// TwinCAT 3 PLC project control
// ProgramVersion: 3.1.4023.0
// libraries:
//   CmpBitmapPool, * (System)
//   Tc2_MC2, * (Beckhoff Automation GmbH)
//   Tc2_ModbusRTU, * (Beckhoff Automation GmbH)
//   Tc2_SerialCom, * (Beckhoff Automation GmbH)
//   Tc2_Standard, * (Beckhoff Automation GmbH)
//   Tc2_System, * (Beckhoff Automation GmbH)
//   Tc2_Utilities, * (Beckhoff Automation GmbH)
//   Tc3_Module, * (Beckhoff Automation GmbH)
//   VisuDialogs, * (System)
//   VisuSymbols,3.5.10.0,System
// project tree:
//   FB/ Rec_Ctrl.TcPOU
//   / GlobalTextList.TcGTLO, ImagePool_Base.TcIPO (not stored), PlcTask.TcTTO, Recipt_no.TcTLO, step.TcTLO, Visualization Manager.TcVMO (not stored), VISU_TASK.TcTTO
//   GVLs/ GVL.TcGVL
//   POUs/ MAIN.TcPOU, MOTION.TcPOU, POU.TcPOU
//   VISUs/ ALARM.TcVIS, IO_TABLE.TcVIS, MainBase.TcVIS, MOTION.TcVIS, PARAMETER.TcVIS, Recipt.TcVIS

CONFIGURATION control
    RESOURCE PLC ON TwinCAT3
        TASK PlcTask(INTERVAL := T#10ms, PRIORITY := 20);
        TASK VISU_TASK(INTERVAL := T#200000us, PRIORITY := 30);
        PROGRAM MAIN WITH PlcTask : MAIN;
        PROGRAM POU WITH PlcTask : POU;
        PROGRAM MOTION WITH PlcTask : MOTION;
        PROGRAM VisuElems_Visu_Prg WITH VISU_TASK : VisuElems.Visu_Prg;
    END_RESOURCE
END_CONFIGURATION

// ---- GVLs/GVL.TcGVL

VAR_GLOBAL
	

DI0_0 AT %I* :BOOL;
DI0_1 AT %I* :BOOL;
DI0_2 AT %I* :BOOL;
DI0_3 AT %I* :BOOL;
DI0_4 AT %I* :BOOL;
DI0_5 AT %I* :BOOL;
DI0_6 AT %I* :BOOL;
DI0_7 AT %I* :BOOL;

DI1_0 AT %I* :BOOL;
DI1_1 AT %I* :BOOL;
DI1_2 AT %I* :BOOL;
DI1_3 AT %I* :BOOL;
DI1_4 AT %I* :BOOL;
DI1_5 AT %I* :BOOL;
DI1_6 AT %I* :BOOL;
DI1_7 AT %I* :BOOL;

DI2_0 AT %I* :BOOL;
DI2_1 AT %I* :BOOL;
DI2_2 AT %I* :BOOL;
DI2_3 AT %I* :BOOL;
DI2_4 AT %I* :BOOL;
DI2_5 AT %I* :BOOL;
DI2_6 AT %I* :BOOL;
DI2_7 AT %I* :BOOL;

DI3_0 AT %I* :BOOL;
DI3_1 AT %I* :BOOL;
DI3_2 AT %I* :BOOL;
DI3_3 AT %I* :BOOL;
DI3_4 AT %I* :BOOL;
DI3_5 AT %I* :BOOL;
DI3_6 AT %I* :BOOL;
DI3_7 AT %I* :BOOL;


DO0_0 AT %Q* :BOOL;
DO0_1 AT %Q* :BOOL;
DO0_2 AT %Q* :BOOL;
DO0_3 AT %Q* :BOOL;
DO0_4 AT %Q* :BOOL;
DO0_5 AT %Q* :BOOL;
DO0_6 AT %Q* :BOOL;
DO0_7 AT %Q* :BOOL;

DO1_0 AT %Q* :BOOL;
DO1_1 AT %Q* :BOOL;
DO1_2 AT %Q* :BOOL;
DO1_3 AT %Q* :BOOL;
DO1_4 AT %Q* :BOOL:=1;
DO1_5 AT %Q* :BOOL:=1;
DO1_6 AT %Q* :BOOL:=1;
DO1_7 AT %Q* :BOOL:=1;

DO2_0 AT %Q* :BOOL;
DO2_1 AT %Q* :BOOL;
DO2_2 AT %Q* :BOOL;
DO2_3 AT %Q* :BOOL;
DO2_4 AT %Q* :BOOL;
DO2_5 AT %Q* :BOOL;
DO2_6 AT %Q* :BOOL;
DO2_7 AT %Q* :BOOL;

DO3_0 AT %Q* :BOOL;
DO3_1 AT %Q* :BOOL;
DO3_2 AT %Q* :BOOL;
DO3_3 AT %Q* :BOOL;
DO3_4 AT %Q* :BOOL;
DO3_5 AT %Q* :BOOL;
DO3_6 AT %Q* :BOOL;
DO3_7 AT %Q* :BOOL;

DO4_0 AT %Q* :BOOL;
DO4_1 AT %Q* :BOOL;
DO4_2 AT %Q* :BOOL;
DO4_3 AT %Q* :BOOL;
DO4_4 AT %Q* :BOOL;
DO4_5 AT %Q* :BOOL;
DO4_6 AT %Q* :BOOL;
DO4_7 AT %Q* :BOOL;

DO5_0 AT %Q* :BOOL;
DO5_1 AT %Q* :BOOL;
DO5_2 AT %Q* :BOOL;
DO5_3 AT %Q* :BOOL;
DO5_4 AT %Q* :BOOL;
DO5_5 AT %Q* :BOOL;
DO5_6 AT %Q* :BOOL;
DO5_7 AT %Q* :BOOL;


AI0_0 AT %I* :UINT;
AI0_1 AT %I* :UINT;
AI0_2 AT %I* :UINT;
AI0_3 AT %I* :UINT;//CG1

AI1_0 AT %I* :UINT;//CG2
AI1_1 AT %I* :UINT;//CG3
AI1_2 AT %I* :UINT;
AI1_3 AT %I* :UINT;

AI2_0 AT %I* :UINT;//temp new add
AI2_1 AT %I* :UINT;
AI2_2 AT %I* :UINT;
AI2_3 AT %I* :UINT;


AO0_0 AT %Q* :UINT;
AO0_1 AT %Q* :UINT;
AO0_2 AT %Q* :UINT;
AO0_3 AT %Q* :UINT;

GV1_CLS_DEVINP: BOOL;
GV1_OPN_DEVINP: BOOL;
GV1_OPN_CONST:REAL:=-10;

GV2_CLS_DEVINP: BOOL;
GV2_OPN_DEVINP: BOOL;
GV2_OPN_CONST:REAL:=10;

MFC1_open_btn:BOOL;
MFC2_open_btn:BOOL;

HTC_SetPos:WORD;
HTC_SetPr:WORD;
Rec_start_btn:BOOL;
Rec_stop_btn:BOOL;

//Recipt variable
lv80_btn: BOOL;
WSU_btn: BOOL;
MFC1_Inp: REAL;
MFC2_Inp: REAL;
GV1_btn_open: BOOL;
GV1_btn_close: BOOL;
GV2_btn_open: BOOL;
GV2_btn_close: BOOL;

SV1 : WORD;
SV2 : WORD;
SV3 : WORD;

Temp_Recipt_step: Recipt_step;

M1TOM2:BOOL;
M2ToM3:BOOL;
M3ToM2:BOOL;
M2ToM1:BOOL;
ON_POS:BOOL;
CUR_step_name:STRING(20);
Rec_finish:BOOL;
ON_POS_FLAG: BOOL;
M2ToM1_flag: BOOL;
M3ToM2_flag: BOOL;
M2ToM3_flag: BOOL;
M1ToM2_flag: BOOL;
swing_btn:BOOL;
take_up_btn:BOOL;
put_down_btn:BOOL;
Rec_take_up_finish:BOOL;
Rec_put_down_finish:BOOL;
M2_pressure_setting:REAL;
M2_current_pressure:real;
END_VAR

// ---- POUs/MAIN.TcPOU
PROGRAM MAIN
VAR
	MbMster: ModbusRtuMaster_KL6x22B;
	Mb_ID: BYTE;
	MbR_Q: WORD;
	MbR_Addr: WORD;
	Data_Read : ARRAY[1..8] OF INT;
	Data_Write : WORD;
	En_Read : BOOL;
    En_Write : BOOL;	
	MbW_Addr: WORD;
	
	PV1 : INT;
	PV2 : INT;
	PV3 : INT;
	
	
	
	nVar: INT;
	bVar1: BOOL;
	bVar3: BOOL;
	bVar2: BOOL;
	
	TTR91_U_CG1: LREAL;
	TTR91_P_CG1: LREAL;
	TTR91_C: REAL:=6.304;
	temp_CG1: LREAL;
	temp_string_CG1:STRING(255);
	strlen_CG1:INT;
	str1_CG1:STRING(255);
	str2_CG1:STRING(255);
	show_CG1:STRING(255);
	aSplit_CG1       : ARRAY[1..5] OF STRING(255);
	bResultSplit_CG1 : BOOL;
	i_CG1            : UDINT;
	
	TTR91_U_CG2: LREAL;
	TTR91_P_CG2: LREAL;
	temp_CG2: LREAL;
	temp_string_CG2:STRING(255);
	strlen_CG2:INT;
	str1_CG2:STRING(255);
	str2_CG2:STRING(255);
	show_CG2:STRING(255);
	aSplit_CG2       : ARRAY[1..5] OF STRING(255);
	bResultSplit_CG2 : BOOL;
	i_CG2            : UDINT;
	
	TTR91_U_CG3: LREAL;
	TTR91_P_CG3: LREAL;
	temp_CG3: LREAL;
	temp_string_CG3:STRING(255);
	strlen_CG3:INT;
	str1_CG3:STRING(255);
	str2_CG3:STRING(255);
	show_CG3:STRING(255);
	aSplit_CG3       : ARRAY[1..5] OF STRING(255);
	bResultSplit_CG3 : BOOL;
	i_CG3            : UDINT;
		

	ATM1_dis: REAL;
	ATM2_dis: REAL;
	ATM3_dis: REAL;
	MFC1_dis: REAL;
	MFC2_dis: REAL;
	
	MFC1_Out: UINT;
	MFC2_Out: uINT;
	
	

	
	WSU_DEVINP: BOOL;
	RST_BTN: BOOL;
	ALM_PUMP_COOL: BOOL;
	ALM_MFC1_DEV: BOOL;
	ALM_MFC2_DEV: BOOL;
	ALM_WATER_TEMP: BOOL;
	ALM_WATER_Prs: BOOL;
	ALM_Heater1_Temp:BOOL;
	ALM_Heater2_Temp:BOOL;
	ALM_Heater_cool:BOOL;
	ALM_GV1_Snr:BOOL;
	ALM_GV2_Snr:BOOL;
	ALM_inlet_prs:BOOL;
	
	MFC_ALM_TIMER1:TON;
	MFC_ALM_TIMER2:TON;
	WTR_TEMP_ALM_TIMER:TON;
	WP_IN_ALM_TIMER:Ton;
	WTR_DELTA_ALM_TIMER:Ton;
	HEATER_TEMP_ALM_TIMER1:Ton;
	HEATER_TEMP_ALM_TIMER2:Ton;
	
	MFC_ALM_TRIG1:R_TRIG;
	MFC_ALM_TRIG2:R_TRIG;
	WTR_TEMP_ALM_TRIG:R_TRIG;
	WP_IN_ALM_TRIG:R_TRIG;
	WTR_DELTA_ALM_TRIG:R_TRIG;
	HEATER_TEMP_ALM_TRIG1:R_TRIG;
	HEATER_TEMP_ALM_TRIG2:R_TRIG;
	
	MFC_ALM_FLAG1:BOOL;
	MFC_ALM_FLAG2:BOOL;
	WTR_TEMP_ALM_FLAG:BOOL;
	WP_IN_ALM_FLAG:BOOL;
	WTR_DELTA_ALM_FLAG:BOOL;
	HEATER_TEMP_ALM_FLAG1:BOOL;
	HEATER_TEMP_ALM_FLAG2:BOOL;
	
	
	MFC_delay:TIME;
	water_temp_delay:TIME;
	WP_IN_delay:TIME;
	WP_delta_delay:TIME;
	Heater_temp_delay:TIME;
	
	GV1_DFLAG: BOOL;
	GV1_TON: TON;
	ALM_GV1_CLS_SNR: BOOL;
	GV2_DFLAG: BOOL;
	GV2_TON: TON;
	ALM_GV2_CLS_SNR: BOOL;
	MbMster2: ModbusRtuMaster_KL6x22B;
	Data_Read2:ARRAY[1..8] OF INT;
	MbR_Q2: WORD;
	MbR_Addr2: WORD;
	En_Read2: BOOL;
	nVar2: INT;
	ADDR2: WORD; 
	En_Write2: BOOL;
	MbW_Addr2: WORD;
	Data_Write2: WORD;
	
	m3_up_btn:BOOL;
	m3_down_btn:BOOL;
	m3_rail_open:BOOL;
	m3_rail_cls:BOOL;
	m3_pin_up:BOOL;
	m3_pin_down:BOOL;
	
	m3_up_flag: BOOL;
	m3_down_flag: BOOL;
	up_step1: BOOL;
	up_step2: BOOL;
	M3_rail_opened: BOOL;
	up_step3: BOOL;
	up_step4: BOOL;
	up_step5: BOOL;
	down_step1: BOOL;
	down_step2: BOOL;
	down_step3: BOOL;
	down_step4: BOOL;
	M3_rail_closed: BOOL;
	HTC_ReadPos: INT;
	HTC_ReadPr: INT;
	//HTC_SetPr: WORD;
	HTC_MODE_Pr : BOOL;
	//HTC_SetPos: WORD;
	
	cur_mode:STRING(255);
	
	M1_sNR: BOOL;
	M2_SNR1: BOOL;
	M2_SNR2: BOOL;
	M3_SNR1: BOOL;
	M3_SNR2: BOOL;
	M3_SNR3: BOOL;
	mfc1_set: REAL;
	mfc2_set: REAL;
	M3_rail_CLOSE: BOOL;
	ATM1_STS: BOOL;
	ATM2_STS: BOOL;
	ATM3_STS: BOOL;
	LV80_STS: BOOL;
	WSU_STS: bool;
	TV_STS: BOOL;
	
	GetTime:NT_GetTime;
	cur_time:STRING(255);
	
	reset_btn:BOOL;
	insert_btn:bool;

	Rec_Ctrl:Rec_Ctrl;
	Copy_step:BOOL;
	Copy_recipe:BOOL;
	cur_step:INT:=1;
	cur_Rec:INT:=1;
	
	save_step_btn: BOOL;
	clear_step_btn:BOOL;
	//edit_step_btn:BOOL;	
	pre_step:INT:=1;
	pre_recipe:INT:=1;
	Rec_finish_delay: TON;
	Rec_finish_trig: R_TRIG;
	take_up_action: BOOL;
	put_down_action: BOOL;
	Rec_stop: BOOL;
	Rec_stop_btn_delay: TON;
	put_down_reset_action: TON;
	put_down_action_reset_in: BOOL;
	take_up_action_reset_in: BOOL;
	take_up_reset_action: TON;
	i: INT;
	j: INT;
	recipe_varible_reset_btn: BOOL;

	q: INT:=30;
	insert_delay:TON;
	insert_in:BOOL;
	insert_during: BOOL;
	insert_finish: BOOL;
END_VAR


VAR RETAIN
    MFC_delay_show:UINT;
	water_temp_delay_show:UINT;
	WP_IN_delay_show:UINT;
	WP_delta_delay_show:UINT;
	Heater_temp_delay_show:UINT;
	MFC_alarm_setting:REAL;
	water_temp_setting:REAL;
	WP_IN_setting:REAL;
	WP_delta_setting:REAL;
	Heater_temp_seeting:REAL;
	Full_recipt: ARRAY [1..10] OF One_Recipt;
END_VAR

CASE nVar OF 
     0 : 
		 En_Read := FALSE;
         En_Write := FALSE;	 
         IF NOT MbMster.BUSY AND NOT En_Write THEN
		   nVar := 1;	
		 END_IF
	 1 :
	     Mb_ID := 1;
		 MbR_Q := 1;
		 MbR_Addr := 130;
		 En_Read := TRUE;
         IF NOT MbMster.BUSY AND En_Read THEN
		   PV3 := MAIN.Data_Read[1]; 
		   nVar := 2;	
		 END_IF

     2 : 
	 
		 En_Read := FALSE;
         En_Write := FALSE;
         IF NOT MbMster.BUSY AND NOT En_Read  THEN
		   nVar := 3;	
		 END_IF
	 3 :
	     Mb_ID := 2;
		 MbR_Q := 1;
		 MbR_Addr := 130;
		 En_Read := TRUE;
         IF NOT MbMster.BUSY AND En_Read  THEN
		   PV1 := MAIN.Data_Read[1];				 
		   nVar := 4;	
		 END_IF	    
     4 : 

		 En_Read := FALSE;
         En_Write := FALSE;
         IF NOT MbMster.BUSY AND NOT En_Read  THEN
		   nVar := 5;	
		 END_IF
	 5 :
	     Mb_ID := 3;
		 MbR_Q := 1;
		 MbR_Addr := 130;
		 En_Read := TRUE;
         IF NOT MbMster.BUSY AND En_Read  THEN
		   PV2 := MAIN.Data_Read[1];			 
		   nVar := 6;	
		 END_IF	 
     6 : 
	 
         MAIN.Data_Write := SV1;		 
		 En_Read := FALSE;
         En_Write := FALSE;
         IF NOT MbMster.BUSY AND NOT En_Read  THEN
		   nVar := 7;	
		 END_IF
	 7 :
	     Mb_ID := 1;
		 MbW_Addr := 49;
		 En_Write := TRUE;
         IF NOT MbMster.BUSY AND En_Write  THEN
		   nVar := 8;	
		 END_IF
     8 : 
		 En_Read := FALSE;
         En_Write := FALSE;
         MAIN.Data_Write := SV2;		 
         IF NOT MbMster.BUSY  AND NOT En_Write  THEN
		   nVar := 9;	
		 END_IF
	 9 :
	     Mb_ID := 2;
		 MbW_Addr := 49;
		 En_Write := TRUE;
         IF NOT MbMster.BUSY  AND En_Write  THEN
		   nVar := 10;	
		 END_IF
     10 : 
		 En_Read := FALSE;
         En_Write := FALSE;
		 MAIN.Data_Write := SV3;
         IF NOT MbMster.BUSY  AND NOT En_Write  THEN
		   nVar := 11;	
		 END_IF
	 11 :
	     Mb_ID := 3;
		 MbW_Addr := 49;
		 En_Write := TRUE;
         IF NOT MbMster.BUSY  AND En_Write  THEN
		   nVar := 0;	
		 END_IF  	 


//ELSE 
		 //nVar := 0;
         //bVar1 := NOT bVar1; 
         //bVar2 := bVar1 OR bVar2; 
END_CASE;	


MbMster.ReadRegs(
	UnitID:= Mb_ID, 
	Quantity:= MbR_Q,
	MBAddr:= MbR_Addr, 
	cbLength:= SIZEOF(Data_Read), 
	pMemoryAddr:= ADR(Data_Read), 
	Execute:= En_Read, 
	Timeout:= T#10S, 
	BUSY=> , 
	Error=> , 
	ErrorId=> , 
	cbRead=> );

MbMster.WriteRegs(
	UnitID:= Mb_ID, 
	Quantity:= 1, 
	MBAddr:= MbW_Addr, 
	cbLength:= SIZEOF(Data_Write), 
	pMemoryAddr:= ADR(Data_Write), 
	Execute:= En_Write, 
	Timeout:= T#10S, 
	BUSY=> , 
	Error=> , 
	ErrorId=> , 
	cbRead=> );	
	
//============= RS485 CH2	

CASE nVar2 OF 
     0 : 
		 En_Read2 := FALSE;
         En_Write2 := FALSE;	 
         IF NOT MbMster2.BUSY  AND NOT En_Read2 THEN
		   nVar2 := 1;	
		 END_IF
	 1 :
	     //Mb_ID := 1;
		 MbR_Q2 := 1;
		 MbR_Addr2 := 263;//259;
		 En_Read2 := TRUE;
         IF NOT MbMster2.BUSY  AND   En_Read2 THEN
			 HTC_ReadPos := MAIN.Data_Read2[1];
		     nVar2 := 2;	
		 END_IF
	 2 : 
	   	 //MbW_Addr2 := WADDR2;
		 En_Read2 := FALSE;
		 En_Write2 := FALSE;
         IF NOT MbMster2.BUSY AND NOT En_Read2 THEN
		   nVar2 := 3;	
		 END_IF
	 3 :
	     //Mb_ID := 1;
		 //MbR_Q2 := 1;
		 IF HTC_MODE_Pr THEN
			HTC_SetPos :=0; 
		 END_IF
		 MAIN.Data_Write2 := HTC_SetPos;
		 MbW_Addr2 := 260;
		 En_Write2 := TRUE;
         IF NOT MbMster2.BUSY  AND   En_Write2 THEN
		     nVar2 := 4;	
		 END_IF
	 4 : 
	   	 //MbW_Addr2 := WADDR2;
		 En_Read2 := FALSE;
		 En_Write2 := FALSE;
         IF NOT MbMster2.BUSY AND NOT En_Write2 THEN
		   nVar2 := 5;	
		 END_IF		 		 
	 5 :
	     //Mb_ID := 1;
		 MbR_Q2 := 1;
		 MbR_Addr2 := 259;//263;
		 En_Read2 := TRUE;
         IF NOT MbMster2.BUSY  AND   En_Read2 THEN
			 HTC_ReadPr := MAIN.Data_Read2[1];
		     nVar2 := 6;	
		 END_IF
	 6 : 
	   	 //MbW_Addr2 := WADDR2;
		 En_Read2 := FALSE;
		 En_Write2 := FALSE;
         IF NOT MbMster2.BUSY AND NOT En_Read2 THEN
		   nVar2 := 7;	
		 END_IF
	 7 :
	     //Mb_ID := 1;
		 //MbR_Q2 := 1;
		 IF NOT HTC_MODE_Pr THEN
			 HTC_SetPr := 0;
		 END_IF
		 MAIN.Data_Write2 := HTC_SetPr;
		 MbW_Addr2 := 1123;
		 En_Write2 := TRUE;
         IF NOT MbMster2.BUSY  AND   En_Write2 THEN
		     nVar2 := 8;	
		 END_IF
	 8 : 
	   	 //MbW_Addr2 := WADDR2;
		 En_Read2 := FALSE;
		 En_Write2 := FALSE;
         IF NOT MbMster2.BUSY AND NOT En_Write2 THEN
		   nVar2 := 0;	
		 END_IF		 		 
		 
END_CASE;


MbMster2.ReadRegs(
	UnitID:= 1, 
	Quantity:= MbR_Q2, 
	MBAddr:= MbR_Addr2, 
	cbLength:= SIZEOF(Data_Read2), 
	pMemoryAddr:= ADR(Data_Read2), 
	Execute:= En_Read2, 
	Timeout:= T#10S, 
	BUSY=> , 
	Error=> , 
	ErrorId=> , 
	cbRead=> );

	MbMster2.WriteRegs(
	UnitID:= 1, 
	Quantity:= 1, 
	MBAddr:= MbW_Addr2, 
	cbLength:= SIZEOF(Data_Write2), 
	pMemoryAddr:= ADR(Data_Write2), 
	Execute:= En_Write2, 
	Timeout:= T#10S, 
	BUSY=> , 
	Error=> , 
	ErrorId=> , 
	cbRead=> );	


//=========================
CG1_trans();
CG2_trans();
CG3_trans();
interlock();
valve_control();
//ALARM();
snr_status();


IF insert_btn  = 1  THEN
	step_insert();
END_IF

IF insert_finish THEN
	insert_btn:=0;
	insert_finish:=0;
END_IF

IF Rec_stop_btn THEN
	Rec_stop:=1;
	REC_func();	
END_IF
Rec_stop_btn_delay(IN:=Rec_stop,PT:=T#0.1S,Q=>);
IF Rec_stop_btn_delay.Q THEN
	REC_func();	
	Rec_stop:=0;
	Rec_finish:=1;
END_IF

IF Rec_start_btn THEN
	REC_func();
END_IF

IF Rec_finish = 1 THEN
	Rec_reset();	
END_IF

IF Rec_finish_trig.Q THEN
	Rec_finish:=0;
END_IF

Rec_finish_delay(IN:=Rec_finish,PT:=T#0.1S,Q=>);
Rec_finish_trig(CLK:=Rec_finish_delay.Q,Q=>);

//ATM

	ATM1_dis:= 100*((UINT_TO_REAL(ai0_0)-19660)/13106);
	ATM2_dis:= 100*((UINT_TO_REAL(ai0_1)-19660)/13106);
	ATM3_dis:= 100*((UINT_TO_REAL(ai0_2)-19660)/13106);

//MFC1 1SLM  MFC 100SLM

    MFC1_dis:=1000*(UINT_TO_REAL(ai1_2)/32767);
	MFC2_dis:=100*(UINT_TO_REAL(ai1_3)/32767);	
	
	IF mfc1_open_btn THEN     //2022 0923 modify
		mfc1_set:=MFC1_Inp;
		ELSE
		mfc1_set:=0;
	END_IF
	
	IF mfc2_open_btn THEN
		mfc2_set:=MFC2_Inp;
		ELSE
		mfc2_set:=0;
	END_IF
	
	MFC1_Out:=REAL_TO_UINT(mfc1_set/1000*32767);
	MFC2_Out:=REAL_TO_UINT(mfc2_set/100*32767);
	ao0_2:=MFC1_Out;
    ao0_3:=MFC2_Out;
	
IF HTC_MODE_Pr = 1 THEN
	cur_mode:='Pos mode';
ELSE
	cur_mode:='Pr mode';
END_IF

IF GetTime.START AND NOT GetTime.BUSY THEN
	GetTime.START:=FALSE;
ELSE
	GetTime.START:=TRUE;
END_IF

GetTime(
	NETID:= '',
	START:= ,
	TMOUT:= ,
	BUSY=> ,
	ERR=>,
	ERRID=>,
	TIMESTR=>
);
cur_time:=CONCAT(WORD_TO_STRING(GetTime.TIMESTR.wHour),':');
cur_time:=CONCAT(cur_time,WORD_TO_STRING(GetTime.TIMESTR.wMinute));
cur_time:=CONCAT(cur_time,':');
cur_time:=CONCAT(cur_time,WORD_TO_STRING(GetTime.TIMESTR.wSecond));

IF save_step_btn THEN
	pre_step:=cur_step;
	pre_recipe:=cur_REC;
	Full_Recipt[cur_Rec].Rec_array[cur_step]:=Temp_Recipt_step;
END_IF

IF pre_step <> cur_step THEN
	Temp_Recipt_step:=Full_Recipt[cur_Rec].Rec_array[cur_step];
	pre_step:=cur_step;
END_IF

IF pre_recipe <> cur_REC THEN
	Temp_Recipt_step:=Full_Recipt[cur_Rec].Rec_array[cur_step];
	pre_recipe:=cur_rec;
END_IF

IF Copy_step AND cur_Step <> 1 THEN
	Temp_Recipt_step:=Full_Recipt[cur_Rec].Rec_array[cur_step-1];
END_IF

IF Copy_recipe AND cur_Rec <> 1 THEN
	Full_Recipt[cur_Rec]:=Full_Recipt[cur_Rec-1];
	Temp_Recipt_step:=Full_Recipt[cur_Rec].Rec_array[cur_step];
END_IF

IF clear_step_btn = 1 THEN
	Temp_Recipt_step.delay:=0;
	Temp_Recipt_step.GV1:=0;
	Temp_Recipt_step.GV2:=0;
	Temp_Recipt_step.LV80:=0;
	Temp_Recipt_step.M1toM2:=0;
	Temp_Recipt_step.M2_pressure_setting:=0;
	Temp_Recipt_step.M2toM1:=0;
	Temp_Recipt_step.M2toM3:=0;
	Temp_Recipt_step.M3_pressure_setting:=0;
	Temp_Recipt_step.M3toM2:=0;
	Temp_Recipt_step.MFC1_button:=0;
	Temp_Recipt_step.MFC1_Setting:=0;
	Temp_Recipt_step.MFC2_button:=0;
	Temp_Recipt_step.MFC2_Setting:=0;
	Temp_Recipt_step.NC1:=0;
	Temp_Recipt_step.NC2:=0;
	Temp_Recipt_step.NC3:=0;
	Temp_Recipt_step.NC4:=0;
	Temp_Recipt_step.NC5:=0;
	Temp_Recipt_step.NC6:=0;
	Temp_Recipt_step.NC7:=0;
	Temp_Recipt_step.NC8:=0;
	Temp_Recipt_step.NC9:=0;
	Temp_Recipt_step.Position_setting:=0;
	Temp_Recipt_step.RV1:=0;
	Temp_Recipt_step.RV2:=0;
	Temp_Recipt_step.Set2Pos:=0;
	Temp_Recipt_step.step_Name:='';
	Temp_Recipt_step.VENT2:=0;
	Temp_Recipt_step.WSU251:=0;
	Temp_Recipt_step.Swing:=0;
	Temp_Recipt_step.Take_up:=0;
	Temp_Recipt_step.Put_down:=0;
	Temp_Recipt_step.VB4:=0;
	Temp_Recipt_step.VENT3:=0;
END_IF
(*
IF edit_step_btn THEN
	Temp_Recipt_step:=Full_Recipt[cur_Rec].Rec_array[cur_step];
END_IF
*)

IF Rec_stop_btn THEN
	Rec_start_btn:=0;
END_IF

IF recipe_varible_reset_btn THEN
	Recipe_variable_reset();
END_IF

M2_current_pressure:=ATM1_dis;

ACTION ALARM:
//PUMP COOLING WATER

IF DO3_6 AND NOT di1_4 THEN	
	ALM_PUMP_COOL:=1;
END_IF



// inlet pressure

IF NOT di1_7 THEN 
	ALM_inlet_prs:=1;
	ELSE
	ALM_inlet_prs:=0;	
END_IF



//GV1
IF GV1_btn_close THEN
	GV1_DFLAG:=1;
END_IF

GV1_TON(IN:=GV1_DFLAG,PT:=T#3S,Q=>,ET=>);
IF GV1_TON.Q AND NOT DI2_0 THEN
	ALM_GV1_CLS_SNR:=1;
END_IF

IF GV1_btn_OPEN THEN
	GV1_DFLAG:=0;
END_IF


//GV2

IF GV2_btn_close THEN
	GV2_DFLAG:=1;
END_IF

GV2_TON(IN:=GV2_DFLAG,PT:=T#3S,Q=>,ET=>);
IF GV2_TON.Q AND NOT DI2_2 THEN
	ALM_GV2_CLS_SNR:=1;
END_IF

IF GV2_btn_OPEN THEN
	GV2_DFLAG:=0;
END_IF



//Light Tower

IF ALM_PUMP_COOL OR ALM_inlet_prs OR ALM_GV1_CLS_SNR OR ALM_GV2_CLS_SNR THEN
	DO1_4:=0;
	DO1_7:=0;
END_IF



// RST BUTTON
IF RST_BTN THEN
	DO1_4:=1;
	DO1_7:=1;
	ALM_PUMP_COOL:=0;
	ALM_inlet_prs:=0;
	ALM_GV1_CLS_SNR:=0;
	ALM_GV2_CLS_SNR:=0;
END_IF

//alarm delay setting
MFC_delay:=UINT_TO_TIME(MFC_delay_show)*1000;
water_temp_delay:=UINT_TO_TIME(water_temp_delay_show)*1000;
WP_IN_delay:=UINT_TO_TIME(WP_IN_delay_show)*1000;
WP_delta_delay:=UINT_TO_TIME(WP_delta_delay_show)*1000;
Heater_temp_delay:=UINT_TO_TIME(Heater_temp_delay_show)*1000;

MFC_ALM_TIMER1(IN:=MFC_ALM_FLAG1,PT:=MFC_delay,Q=>);
MFC_ALM_TIMER2(IN:=MFC_ALM_FLAG2,PT:=MFC_delay,Q=>);
WTR_TEMP_ALM_TIMER(IN:=WTR_TEMP_ALM_FLAG,PT:=water_temp_delay,Q=>);
WP_IN_ALM_TIMER(IN:=WP_IN_ALM_FLAG,PT:=WP_IN_delay,Q=>);
WTR_DELTA_ALM_TIMER(IN:=WTR_DELTA_ALM_FLAG,PT:=WP_delta_delay,Q=>);
HEATER_TEMP_ALM_TIMER1(IN:=HEATER_TEMP_ALM_FLAG1,PT:=Heater_temp_delay,Q=>);
HEATER_TEMP_ALM_TIMER2(IN:=HEATER_TEMP_ALM_FLAG2,PT:=Heater_temp_delay,Q=>);

MFC_ALM_TRIG1(CLK:=MFC_ALM_TIMER1.Q,Q=>);
MFC_ALM_TRIG2(CLK:=MFC_ALM_TIMER2.Q,Q=>);
WTR_TEMP_ALM_TRIG(CLK:=WTR_TEMP_ALM_TIMER.Q,Q=>);
WP_IN_ALM_TRIG(CLK:=WP_IN_ALM_TIMER.Q,Q=>);
WTR_DELTA_ALM_TRIG(CLK:=WTR_DELTA_ALM_TIMER.Q,Q=>);
HEATER_TEMP_ALM_TRIG1(CLK:=HEATER_TEMP_ALM_TIMER1.Q,Q=>);
HEATER_TEMP_ALM_TRIG2(CLK:=HEATER_TEMP_ALM_TIMER2.Q,Q=>);

IF (MFC1_Inp < MFC1_dis *(1-MFC_alarm_setting*0.01) OR MFC1_Inp > MFC1_dis *(1+MFC_alarm_setting*0.01)) AND MFC1_Inp <> 0 THEN
	MFC_ALM_FLAG1:=1;
	ALM_MFC1_DEV:=1;
ELSE
	MFC_ALM_FLAG1:=0;
	ALM_MFC1_DEV:=0;
END_IF

IF (MFC2_Inp < MFC2_dis *(1-MFC_alarm_setting*0.01) OR MFC2_Inp > MFC2_dis *(1+MFC_alarm_setting*0.01)) AND MFC2_Inp <> 0 THEN
	MFC_ALM_FLAG2:=1;
	ALM_MFC2_DEV:=1;
ELSE
	MFC_ALM_FLAG2:=0;
	ALM_MFC2_DEV:=0;
END_IF

IF MFC_ALM_TRIG1.Q OR MFC_ALM_TRIG2.Q THEN
	DO1_7:=0;//DO1_7:=0會叫
END_IF


IF PV1 > Heater_temp_seeting THEN
	HEATER_TEMP_ALM_FLAG1:=1;
	ALM_Heater1_Temp:=1;
ELSE
	HEATER_TEMP_ALM_FLAG1:=0;
	ALM_Heater1_Temp:=0;
END_IF

IF PV2 > Heater_temp_seeting THEN
	HEATER_TEMP_ALM_FLAG2:=1;
	ALM_Heater2_Temp:=1;
ELSE
	HEATER_TEMP_ALM_FLAG2:=0;
	ALM_Heater2_Temp:=0;
END_IF

IF HEATER_TEMP_ALM_TRIG1.Q OR HEATER_TEMP_ALM_TRIG2.Q THEN
	DO1_7:=0;
END_IF
END_ACTION

ACTION CG1_trans:
TTR91_U_CG1 := AI0_3/6553.5 ;
temp_CG1 := (TTR91_U_CG1 - TTR91_C)/1.286;
TTR91_P_CG1 := EXPT(10,temp_CG1);
IF TTR91_P_CG1 > 1 THEN
	temp_string_CG1 := LREAL_TO_STRING(TTR91_P_CG1);
	aSplit_CG1[1] := temp_string_CG1;
	FOR i_CG1:=1 TO 5 DO
    bResultSplit_CG1 := FindAndSplitChar( sSeparatorChar := '.',  pSrcString := ADR(aSplit_CG1[i_CG1]), 
                                      pLeftString    := ADR(aSplit_CG1[i_CG1]),   nLeftSize  := SIZEOF(aSplit_CG1[i_CG1]), 
                                      pRightString   := ADR(aSplit_CG1[i_CG1+1]), nRightSize := SIZEOF(aSplit_CG1[i_CG1+1]),
                                      bSearchFromRight := FALSE );
    IF NOT bResultSplit_CG1 THEN
        EXIT;
    END_IF
	END_FOR
	str2_CG1:=left(temp_string_CG1,3);
	IF TTR91_P_CG1 >= 100 THEN
		str2_CG1:=REAL_TO_STRING(STRING_TO_INT(str2_CG1)/100.0);
	ELSIF TTR91_P_CG1 < 100 AND TTR91_P_CG1 >= 10 THEN
		str2_CG1:=REAL_TO_STRING(STRING_TO_INT(str2_CG1)/10.0);
	ELSIF TTR91_P_CG1 >=1 AND TTR91_P_CG1 < 10 THEN
		str2_CG1:=REAL_TO_STRING(STRING_TO_real(str2_CG1));
	END_IF
	
	str1_CG1:=CONCAT('e+',INT_TO_STRING(len(aSplit_CG1[1])-1));
	show_CG1 := CONCAT (str2_CG1,str1_CG1);
ELSE
	temp_string_CG1 := LREAL_TO_STRING(TTR91_P_CG1);
	str1_CG1:=right(temp_string_CG1,3);
	str2_CG1:=left(temp_string_CG1,4);
	show_CG1 := CONCAT (str2_CG1,str1_CG1);
END_IF
END_ACTION

ACTION CG2_trans:
TTR91_U_CG2 := AI1_0/6553.5 ;
temp_CG2 := (TTR91_U_CG2 - TTR91_C)/1.286;
TTR91_P_CG2 := EXPT(10,temp_CG2);
IF TTR91_P_CG2 > 1 THEN
	temp_string_CG2 := LREAL_TO_STRING(TTR91_P_CG2);
	aSplit_CG2[1] := temp_string_CG2;
	FOR i_CG2:=1 TO 5 DO
    bResultSplit_CG2 := FindAndSplitChar( sSeparatorChar := '.',  pSrcString := ADR(aSplit_CG2[i_CG2]), 
                                      pLeftString    := ADR(aSplit_CG2[i_CG2]),   nLeftSize  := SIZEOF(aSplit_CG2[i_CG2]), 
                                      pRightString   := ADR(aSplit_CG2[i_CG2+1]), nRightSize := SIZEOF(aSplit_CG2[i_CG2+1]),
                                      bSearchFromRight := FALSE );
    IF NOT bResultSplit_CG2 THEN
        EXIT;
    END_IF
	END_FOR
	str2_CG2:=left(temp_string_CG2,3);
	IF TTR91_P_CG2 >= 100 THEN
		str2_CG2:=REAL_TO_STRING(STRING_TO_INT(str2_CG2)/100.0);
	ELSIF TTR91_P_CG2 < 100 AND TTR91_P_CG2 >=10 THEN
		str2_CG2:=REAL_TO_STRING(STRING_TO_INT(str2_CG2)/10.0);
	ELSIF TTR91_P_CG2 <10 AND TTR91_P_CG2 >=1 THEN
		 str2_CG2:=REAL_TO_STRING(STRING_TO_REAL(str2_CG2));
	END_IF
	
	str1_CG2:=CONCAT('e+',INT_TO_STRING(len(aSplit_CG2[1])-1));
	show_CG2 := CONCAT (str2_CG2,str1_CG2);
ELSE
	temp_string_CG2 := LREAL_TO_STRING(TTR91_P_CG2);
	str1_CG2:=right(temp_string_CG2,3);
	str2_CG2:=left(temp_string_CG2,4);
	show_CG2 := CONCAT (str2_CG2,str1_CG2);
END_IF
END_ACTION

ACTION CG3_trans:
TTR91_U_CG3 := AI1_1/6553.5 ;
temp_CG3 := (TTR91_U_CG3 - TTR91_C)/1.286;
TTR91_P_CG3 := EXPT(10,temp_CG3);
IF TTR91_P_CG3 > 1 THEN
	temp_string_CG3 := LREAL_TO_STRING(TTR91_P_CG3);
	aSplit_CG3[1] := temp_string_CG3;
	FOR i_CG3:=1 TO 5 DO
    bResultSplit_CG3 := FindAndSplitChar( sSeparatorChar := '.',  pSrcString := ADR(aSplit_CG3[i_CG3]), 
                                      pLeftString    := ADR(aSplit_CG3[i_CG3]),   nLeftSize  := SIZEOF(aSplit_CG3[i_CG3]), 
                                      pRightString   := ADR(aSplit_CG3[i_CG3+1]), nRightSize := SIZEOF(aSplit_CG3[i_CG3+1]),
                                      bSearchFromRight := FALSE );
    IF NOT bResultSplit_CG3 THEN
        EXIT;
    END_IF
	END_FOR
	str2_CG3:=left(temp_string_CG3,3);
	IF TTR91_P_CG3 >= 10 AND TTR91_P_CG3 < 100 THEN
		str2_CG3:=REAL_TO_STRING(STRING_TO_INT(str2_CG3)/10.0);
	ELSIF TTR91_P_CG3 >= 100 THEN
		str2_CG3:=REAL_TO_STRING(STRING_TO_INT(str2_CG3)/100.0);
	ELSIF TTR91_P_CG3 < 10 AND TTR91_P_CG3 >= 1 THEN
		str2_CG3:=REAL_TO_STRING(STRING_TO_REAL(str2_CG3));
	END_IF
	
	str1_CG3:=CONCAT('e+',INT_TO_STRING(len(aSplit_CG3[1])-1));
	show_CG3 := CONCAT (str2_CG3,str1_CG3);
ELSE
	temp_string_CG3 := LREAL_TO_STRING(TTR91_P_CG3);
	str1_CG3:=right(temp_string_CG3,3);
	str2_CG3:=left(temp_string_CG3,4);
	show_CG3 := CONCAT (str2_CG3,str1_CG3);
END_IF
END_ACTION

ACTION INTERLOCK:
//GV1

IF NOT DI0_0 AND NOT DI0_1 THEN
	GV1_CLS_DEVINP:=1;
	ELSE
	GV1_CLS_DEVINP:=0;	
END_IF

IF ATM1_DIS <GV1_OPN_CONST THEN
	GV1_OPN_DEVINP:=1;
	ELSE
	GV1_OPN_DEVINP:=0;	
END_IF

//GV2

IF NOT DI0_2 AND NOT DI0_3 THEN
	GV2_CLS_DEVINP:=1;
	ELSE
	GV2_CLS_DEVINP:=0;	
END_IF

IF ABS(ATM1_DIS-ATM2_DIS)>GV2_OPN_CONST THEN
	GV2_OPN_DEVINP:=1;
	ELSE
	GV2_OPN_DEVINP:=0;	
END_IF

// LV80 Pump

IF LV80_btn AND di1_4 THEN
	DO3_6:=1;
	ELSE
	DO3_6:=0;
	LV80_btn:=0;
END_IF

IF WSU_btn AND DO3_6 THEN
	DO3_7:=1;
	ELSE
	DO3_7:=0;	
END_IF

//wsu_devinp

IF DO3_6 THEN
	WSU_DEVINP:=0;
	ELSE
	WSU_DEVINP:=1;	
END_IF
END_ACTION

ACTION REC_func:
Rec_Ctrl(
	Enable		:= Rec_start_btn,
	Stop        := Rec_stop, 
	Step		:= Full_Recipt[cur_rec], 
	bStart		=> , 
	State       => , 
	bBusy		=> , 
	bDone		=> , 
	bError		=> );
END_ACTION

ACTION Rec_reset:
CUR_step_name:='';
GV1_btn_open:=0;
GV1_btn_close:=0;
GV2_btn_open:=0;
GV2_btn_close:=0;
lv80_btn:=0;
WSU_btn:=0;
MFC1_Inp:=0;
MFC2_Inp:=0;
mfc1_open_btn:=0;
mfc2_open_btn:=0;
DO2_0:=0;
DO2_1:=0;
DO2_2:=0;
DO2_3:=0;
DO2_4:=0;
DO2_5:=0;
DO2_6:=0;
DO2_7:=0;
DO3_0:=0;
DO3_1:=0;
DO3_2:=0;
DO3_3:=0;
DO4_0:=0;
DO4_1:=0;
DO4_2:=0;
DO4_3:=0;
DO4_4:=0;
DO4_5:=0;
DO4_6:=0;
DO4_7:=0;
DO5_0:=0;
ON_POS:=0;
M1TOM2:=0;
M2ToM3:=0;
M3ToM2:=0;
M2ToM1:=0;
ON_POS_FLAG:=0;
M1ToM2_flag:=0;
M2ToM3_flag:=0;
M3ToM2_flag:=0;
M2ToM1_flag:=0;
take_up_btn:=0;
put_down_btn:=0;
swing_btn:=0;
Rec_take_up_finish:=0;
Rec_put_down_finish:=0;
END_ACTION

ACTION Recipe_variable_reset:
FOR i := 1 TO 10 DO
	FOR j := 1 TO 30 DO
		Full_recipt[i].Rec_array[j].step_Name:= WSTRING_TO_STRING("");
		Full_recipt[i].Rec_array[j].GV1:=0;
		Full_recipt[i].Rec_array[j].GV2:=0;
		Full_recipt[i].Rec_array[j].LV80:=0;
		Full_recipt[i].Rec_array[j].M1toM2:=0;
		Full_recipt[i].Rec_array[j].M2_pressure_setting:=0;
		Full_recipt[i].Rec_array[j].M2toM1:=0;
		Full_recipt[i].Rec_array[j].M2toM3:=0;
		Full_recipt[i].Rec_array[j].M3toM2:=0;
		Full_recipt[i].Rec_array[j].MFC1_button:=0;
		Full_recipt[i].Rec_array[j].MFC1_Setting:=0;
		Full_recipt[i].Rec_array[j].MFC2_button:=0;
		Full_recipt[i].Rec_array[j].MFC2_Setting:=0;
		Full_recipt[i].Rec_array[j].NC1:=0;
		Full_recipt[i].Rec_array[j].NC2:=0;
		Full_recipt[i].Rec_array[j].NC3:=0;
		Full_recipt[i].Rec_array[j].NC4:=0;
		Full_recipt[i].Rec_array[j].NC5:=0;
		Full_recipt[i].Rec_array[j].NC6:=0;
		Full_recipt[i].Rec_array[j].NC7:=0;
		Full_recipt[i].Rec_array[j].NC8:=0;
		Full_recipt[i].Rec_array[j].NC9:=0;
		Full_recipt[i].Rec_array[j].Position_setting:=0;
		Full_recipt[i].Rec_array[j].Put_down:=0;
		Full_recipt[i].Rec_array[j].RV1:=0;
		Full_recipt[i].Rec_array[j].RV2:=0;
		Full_recipt[i].Rec_array[j].Set2Pos:=0;
		Full_recipt[i].Rec_array[j].Swing:=0;
		Full_recipt[i].Rec_array[j].Take_up:=0;
		Full_recipt[i].Rec_array[j].VB4:=0;
		Full_recipt[i].Rec_array[j].VENT3:=0;
		Full_recipt[i].Rec_array[j].VENT2:=0;
		Full_recipt[i].Rec_array[j].WSU251:=0;
	END_FOR
	
END_FOR
END_ACTION

ACTION SNR_STATUS:
M1_SNR:=NOT DI0_0;
M2_SNR1:=NOT DI0_1;
M2_SNR2:=NOT DI0_2;
M3_SNR1:=NOT DI0_3;
M3_SNR2:=NOT DI0_4;
M3_SNR3:=NOT DI0_5;

IF ATM1_dis > -10 THEN
	ATM1_STS:=1;
ELSE
	ATM1_STS:=0;
END_IF

IF ATM2_dis > -10 THEN
	ATM2_STS:=1;
ELSE
	ATM2_STS:=0;
END_IF

IF ATM3_dis > -10 THEN
	ATM3_STS:=1;
ELSE
	ATM3_STS:=0;
END_IF

IF DO3_6 THEN
	LV80_STS:=1;
ELSE
	LV80_STS:=0;
END_IF

IF DO3_7 THEN
	WSU_STS:=1;
ELSE
	WSU_STS:=0;
END_IF

IF HTC_ReadPos > 0 THEN
	TV_STS:=1;
ELSE
	TV_STS:=0;
END_IF
END_ACTION

ACTION step_insert:
insert_delay(IN:=insert_in,PT:=T#1MS,Q=>);

IF insert_in = 0 THEN
	insert_in:=1;
END_IF

IF insert_delay.Q AND q > cur_step THEN
	Full_Recipt[cur_Rec].Rec_array[q]:=Full_Recipt[cur_Rec].Rec_array[q-1];
	q:=q-1;
	insert_in:=0;	
END_IF

IF q = cur_step THEN
	Full_Recipt[cur_Rec].Rec_array[cur_step]:=Temp_Recipt_step;
	q:=30;
	insert_finish:=1;
END_IF
END_ACTION

ACTION valve_control:
//GV1 GV2

  IF GV1_btn_open THEN
	  DO1_0:=0;
	  DO1_1:=1;
  END_IF
  
 IF GV1_btn_close THEN
	  DO1_0:=1;
	  DO1_1:=0;
  END_IF 
  
   IF GV2_btn_open THEN
	  DO1_2:=0;
	  DO1_3:=1;
  END_IF
  
 IF GV2_btn_close THEN
	  DO1_2:=1;
	  DO1_3:=0;
  END_IF 
  
  // M3 LOAD 2022/09/23
  
	IF M3_rail_open THEN
	  DO0_0:=0;
	  DO0_1:=1;
	  DO0_4:=0;
	  DO0_5:=1;
	END_IF	 
	
	IF M3_rail_CLOSE THEN  
	  DO0_0:=1;
	  DO0_1:=0;
	  DO0_4:=1;
	  DO0_5:=0;
	END_IF	  
	
	IF M3_pin_up THEN
	  DO0_6:=1;
	  DO0_7:=0;
	  END_IF
	IF M3_pin_DOWN THEN  
	  DO0_6:=0;
	  DO0_7:=1;	  
	END_IF	  

	
	IF di2_5 AND di2_7 AND di3_1 AND di3_3 THEN
		M3_rail_opened:=1;
		ELSE
		M3_rail_opened:=0;	
	END_IF
		IF di2_4 AND di2_6 AND di3_0 AND di3_2 THEN
		M3_rail_closed:=1;
		ELSE
		M3_rail_closed:=0;	
	END_IF 

// up sequence 

 IF m3_up_btn OR (take_up_btn AND NOT take_up_action) THEN
    m3_up_flag:=1;
    m3_down_flag:=0;
    up_step1:=1;
	take_up_action:=1;
 END_IF
 IF m3_up_flag AND up_step1 THEN
    M3_rail_open:=1;
    up_step1:=0;
    up_step2:=1;
 END_IF
 IF m3_up_flag AND up_step2 AND M3_rail_opened THEN
    M3_pin_up:=1;
    up_step2:=0;
    up_step3:=1;
 END_IF
 IF m3_up_flag AND up_step3 AND di3_4 THEN
      M3_rail_open:=0;
   M3_rail_close:=1;//close M3 rail
   up_step3:=0;
   up_step4:=1;
 END_IF
 
 IF m3_up_flag AND up_step4 AND M3_rail_closed  THEN
      M3_pin_up:=0;
   M3_pin_DOWN:=1; // ADD BY HUGO
   up_step4:=0;
   up_step5:=1;
 END_IF
 IF  m3_up_flag AND up_step5 AND  di3_5 THEN
  M3_rail_close:=0;
  up_step5:=0;
  M3_pin_DOWN:=0;
  m3_up_flag:=0;  // ADD BY HUGO
  IF take_up_btn THEN
	  Rec_take_up_finish:=1;
  END_IF
  take_up_action_reset_in:=1;
 END_IF
take_up_reset_action(IN:=take_up_action_reset_in,PT:=T#0.15S,Q=>);
IF take_up_reset_action.Q THEN
	take_up_action:=0;
	take_up_action_reset_in:=0;
END_IF

 
//down sequence
 
 IF (m3_down_btn OR put_down_btn) AND NOT put_down_action THEN
    m3_up_flag:=0;
    m3_down_flag:=1;
    down_step1:=1;
	put_down_action:=1;
 END_IF
 
 IF m3_down_flag AND down_step1 THEN
    M3_pin_up:=1;
    down_step1:=0;
    down_step2:=1;
 END_IF
 
 IF m3_down_flag AND down_step2 AND di3_4 THEN
    M3_rail_open:=1;
    down_step2:=0;
    down_step3:=1;
 END_IF
 IF m3_down_flag AND down_step3 AND m3_rail_opened THEN
    M3_pin_up:=0;
     M3_pin_DOWN:=1; // ADD BY HUGO
    down_step3:=0;
    down_step4:=1;
 END_IF
 IF m3_down_flag AND down_step4 AND di3_5 THEN
    M3_rail_open:=0;
    down_step4:=0;
    m3_down_flag:=0; // ADD BY HUGO
    M3_pin_DOWN:=0;
	IF put_down_btn THEN
		Rec_put_down_finish:=1;
	END_IF
	put_down_action_reset_in:=1;
 END_IF
	
put_down_reset_action(IN:=put_down_action_reset_in,PT:=T#0.15S,Q=>);

IF put_down_reset_action.Q = 1 THEN
	put_down_action:=0;
	put_down_action_reset_in:=0;
END_IF
//reset

IF reset_btn = 1 THEN
	m3_up_btn:=0;
	m3_down_btn:=0;
	m3_down_flag:=0;
	m3_up_flag:=0;
	up_step1:=0;
	up_step2:=0;
	up_step3:=0;
	up_step4:=0;
	up_step5:=0;
	down_step1:=0;
	down_step2:=0;
	down_step3:=0;
	down_step4:=0;
	put_down_action:=0;
	take_up_action:=0;
END_IF

(*	
// up sequence	

	IF m3_up_btn THEN
	   m3_up_flag:=1;
	   m3_down_flag:=0;
	   up_step1:=1;
	END_IF
	IF m3_up_flag AND up_step1 THEN
	   M3_rail_open:=1;
	   up_step1:=0;
	   up_step2:=1;
	END_IF
	IF m3_up_flag AND up_step2 AND M3_rail_opened THEN
	   M3_pin_up:=1;
	   up_step2:=0;
	   up_step3:=1;
	END_IF
	IF m3_up_flag AND up_step3 AND di3_4 THEN
	     M3_rail_open:=0;
		 M3_rail_close:=1;//close M3 rail
		 up_step3:=0;
		 up_step4:=1;
	END_IF
	
	IF m3_up_flag AND up_step4 AND M3_rail_closed  THEN
	     M3_pin_up:=0;
		 up_step4:=0;
		 up_step5:=1;
	END_IF
	IF  m3_up_flag AND up_step5 AND  di3_5 THEN
		M3_rail_close:=0;
		M3_rail_closed:=0;
		up_step5:=0;
	END_IF
	
//down sequence
	
	IF m3_down_btn THEN
	   m3_up_flag:=0;
	   m3_down_flag:=1;
	   down_step1:=1;
	END_IF
	
	IF m3_down_flag AND down_step1 THEN
	   M3_pin_up:=1;
	   down_step1:=0;
	   down_step2:=1;
	END_IF
	
	IF m3_down_flag AND down_step2 AND di3_4 THEN
	   M3_rail_open:=1;
	   down_step2:=0;
	   down_step3:=1;
	END_IF
	IF m3_down_flag AND down_step3 AND m3_rail_opened THEN
	   M3_pin_up:=0;
	   down_step3:=0;
	   down_step4:=1;
	END_IF
	IF m3_down_flag AND down_step4 AND di3_5 THEN
	  down_step4:=0;
    END_IF 
*)
END_ACTION

END_PROGRAM

// ---- FB/Rec_Ctrl.TcPOU
FUNCTION_BLOCK Rec_Ctrl
VAR_INPUT
	Enable     : BOOL;
	Stop       : BOOL;
	Step	   :One_Recipt;
END_VAR
VAR_OUTPUT
	bStart : BOOL;
	bBusy  : BOOL;
	bDone  : BOOL;
	bError : BOOL;
	State  : INT;
END_VAR
VAR
	bTon : BOOL;
	dur : Ton;
	Rec_duration:Ton;
	nState: INT;
	i : INT := 1;
	pos_delay:TON;
	
	M2toM1_delay: Ton;
	M2toM1_in: BOOL;
END_VAR

IF Stop THEN
	bStart := FALSE;
	bBusy  := FALSE;
	bDone  := FALSE;
	bError := FALSE;
	bTon   := FALSE;
	nState := 0;
	i      := 1;
	Rec_finish:=1;
	Stop:=0;
END_IF



CASE nState OF
0 :	
	IF Enable AND NOT (bBusy OR bError) THEN
		bDone  := FALSE;
		bBusy  := TRUE;
		nState := 1;
		i      := 1;
	END_IF
	
	IF NOT Enable THEN
		bBusy  := FALSE;
		bError := FALSE;		
	END_IF	
1 :
	
	IF step.Rec_array[i].delay > 0 THEN //use delay to change step
		bTon   := TRUE;
		bStart := TRUE;	
		
	ELSIF step.Rec_array[i].Set2Pos = 1 THEN //wait until go to right place
		IF (step.Rec_array[i].M1toM2 OR step.Rec_array[i].M3toM2) AND MAIN.M2_SNR1 AND MAIN.M2_SNR2 THEN
			GVL.ON_POS:=1;
		END_IF
		
		IF step.Rec_array[i].M2toM3 AND MAIN.M3_SNR1 AND MAIN.M3_SNR2 THEN
			GVL.ON_POS:=1;
		END_IF
		
		IF step.Rec_array[i].M2toM1 AND main.M2_SNR1 = 0 AND main.M2_SNR2 = 0 THEN
			M2ToM1_in := 1;
			IF M2ToM1_delay.Q THEN
				ON_POS:=1;
			END_IF
		END_IF
		
		IF (Rec_take_up_finish AND take_up_btn) OR (Rec_put_down_finish AND put_down_btn) THEN
			ON_POS:=1;
		END_IF
		
		IF pos_delay.Q THEN
			Rec_take_up_finish:=0;
			Rec_put_down_finish:=0;
			ON_POS:=0;
			M2ToM1_in:=0;
			i:= i + 1;
			nState := 2;
		END_IF
		
	ELSIF step.Rec_array[i].M2_pressure_setting <> 0 THEN
		IF M2_current_pressure > step.Rec_array[i].M2_pressure_setting THEN
			i:= i + 1;
			nState := 2;
		END_IF
		
	ELSE
		i := i + 1;
		IF i > 30 THEN
			i := 1;
			Rec_start_btn:=0;
			Rec_finish:=1;
		END_IF		
	END_IF
	
	IF Rec_duration.Q  AND step.Rec_array[i].Set2Pos = 0 THEN
		i := i + 1;
		IF i > 30 THEN
			i := 1;
		END_IF
		nState := 2;
	END_IF

2 :	
	IF i < 2 THEN
		bDone  := TRUE;
		bBusy  := FALSE;
		nState := 0;
	ELSE
		nState := 1;	
	END_IF
	bStart := FALSE;
	bTon   := FALSE;
END_CASE

Rec_duration(IN:= bTon, PT:= INT_TO_TIME(Step.Rec_array[i].delay)*1000, Q=> , ET=> );//add 0.1s in order to let other delay 
pos_delay(IN:=GVL.ON_POS,PT:=T#0.1S,Q=>);
M2toM1_delay(IN:=M2toM1_in, PT:=T#10S,Q=>);
State := i;

//SV1:=step.Rec_array[i].Heater_Temp1;
//SV2:=step.Rec_array[i].Heater_Temp2;

lv80_btn := step.Rec_array[i].LV80;
WSU_btn := step.Rec_array[i].WSU251;
IF step.Rec_array[i].VB4 = 0 THEN
	DO4_6:=0;
ELSE
	DO4_6:=1;
END_IF

IF step.Rec_array[i].GV1 = 0 THEN
	GV1_btn_close:=1;
	GV1_btn_open:=0;
ELSE
	GV1_btn_close:=0;
	GV1_btn_open:=1;
END_IF

IF step.Rec_array[i].GV2 = 0 THEN
	GV2_btn_open:=0;
	GV2_btn_close:=1;
ELSE
	GV2_btn_open:=1;
	GV2_btn_close:=0;
END_IF

IF step.Rec_array[i].NC1 THEN
	DO2_0:=1;
ELSE
	DO2_0:=0;
END_IF

IF step.Rec_array[i].NC2 THEN
	DO2_1:=1;
ELSE
	DO2_1:=0;
END_IF

IF step.Rec_array[i].NC3 THEN
	DO2_2:=1;
ELSE
	DO2_2:=0;
END_IF

IF step.Rec_array[i].NC4 THEN
	DO2_3:=1;
ELSE
	DO2_3:=0;
END_IF

IF step.Rec_array[i].NC5 THEN
	DO2_4:=1;
ELSE
	DO2_4:=0;
END_IF

IF step.Rec_array[i].NC6 THEN
	DO2_5:=1;
ELSE
	DO2_5:=0;
END_IF

IF step.Rec_array[i].NC7 THEN
	DO2_6:=1;
ELSE
	DO2_6:=0;
END_IF

IF step.Rec_array[i].NC8 THEN
	DO2_7:=1;
ELSE
	DO2_7:=0;
END_IF

IF step.Rec_array[i].NC9 THEN
	DO3_0:=1;
ELSE
	DO3_0:=0;
END_IF

IF step.Rec_array[i].RV1 THEN
	DO4_7:=1;
ELSE
	DO4_7:=0;
END_IF

IF step.Rec_array[i].RV2 THEN
	DO5_0:=1;
ELSE
	DO5_0:=0;
END_IF

IF step.Rec_array[i].VENT2 THEN
	DO4_1:=1;
ELSE
	DO4_1:=0;
END_IF

IF step.Rec_array[i].VENT3 THEN
	DO4_2:=1;
ELSE
	DO4_2:=0;
END_IF

IF step.Rec_array[i].MFC1_button THEN
	mfc1_open_btn:=1;
ELSE
	mfc1_open_btn:=0;
END_IF

IF step.Rec_array[i].MFC2_button THEN
	mfc2_open_btn:=1;
ELSE
	mfc2_open_btn:=0;
END_IF

MFC1_Inp:=step.Rec_array[i].MFC1_Setting;
MFC2_Inp:=step.Rec_array[i].MFC2_Setting;
M1TOM2:=step.Rec_array[i].M1toM2;
M2ToM3:=step.Rec_array[i].M2toM3;
M3ToM2:=step.Rec_array[i].M3toM2;
M2ToM1:=step.Rec_array[i].M2toM1;
HTC_SetPos:=step.Rec_array[i].Position_setting;
CUR_step_name:=step.Rec_array[i].step_Name;
swing_btn:=step.Rec_array[i].Swing;
take_up_btn:=step.Rec_array[i].Take_up;
put_down_btn:=step.Rec_array[i].Put_down;

END_FUNCTION_BLOCK

// ---- POUs/POU.TcPOU
PROGRAM POU
VAR
    bStart          : BOOL := TRUE;
    fbTimer         : TON;
    tTimerValue     : TIME := T#1S;
    fbTrigger       : R_TRIG;
    tTimeReturn1    : TIME;
    tTimeReturn2    : TIME;
    tDifference     : TIME;	
END_VAR

fbTimer(IN := bStart, PT := tTimerValue);
fbTrigger(CLK := fbTimer.IN);

IF fbTrigger.Q THEN
    tTimeReturn1  := TIME();
END_IF

IF fbTimer.Q THEN
    bStart        := FALSE;
    tTimeReturn2  := TIME();
    tDifference   := tTimeReturn2 - tTimeReturn1;    // The difference will be T#5s
END_IF

END_PROGRAM

// ---- POUs/MOTION.TcPOU
PROGRAM MOTION
VAR
	init: BOOL;
	Power_1: MC_Power;
	Axis1: AXIS_REF;
	Power_2: MC_Power;
	Axis2: AXIS_REF;
	Power_3: MC_Power;
	Axis3: AXIS_REF;
	
	Pwr_En_1: BOOL;
	Pwr1_Err: BOOL;
	Pwr1_ErrId: UDINT;
	MoveStop_1: MC_Stop;
	MoveStop_2: MC_Stop;
	MoveStop_3: MC_Stop;
	stop_1: BOOL;
	Axis1_Speed: INT;
	Axis: INT;
	Execute: INT;
	Deceleration: INT;
	Jerk: INT;
	Options: INT;
	Done: INT;
	Busy: INT;
	Active: INT;
	CommandAborted: INT;
	Error: INT;
	ErrorID: BOOL;
	MoveReset_1: INT;
	reset_1: BOOL;
	Jog_1: MC_Jog;

	AxisReset_1: MC_Reset;
	AxisReset_2: MC_Reset;
	AxisReset_3: MC_Reset;
	JForward: BOOL;
	JBackward: BOOL;
	EN_P: BOOL;
	EN_N: BOOL;
	Jv: LREAL;
	JAcc: LREAL;
	JDec: LREAL;
	Jjerk: LREAL;
	MoveVelocity_1: MC_MoveVelocity;
	MoveVelocity_2: MC_MoveVelocity;
	MoveVelocity_3: MC_MoveVelocity;
	V_ex: BOOL;
	VV: LREAL;
	Halt_1: MC_Halt;
	H_ex: BOOL;
	MoveRelative_1: MC_MoveRelative;
	R_ex: BOOL;
	R_v: LREAL;
	R_dis: LREAL;
	Move_Absolute_1: MC_MoveAbsolute;
	A_ex: BOOL;
	A_pos: LREAL;
	A_v: LREAL;
	DIR1: bool;
	VV1: LREAL:=100;
	V_ex1: BOOL;

	Pwr_En_2: BOOL;
	stop_2: BOOL;
	Axis2_Speed: INT;
	reset_2: BOOL;
	V_ex2: BOOL;
	VV2: LREAL:=100;
	Pwr_En_3: BOOL;
	stop_3: BOOL;
	Axis3_Speed: INT;
	reset_3: BOOL;
	V_ex3: BOOL;
	VV3: LREAL:=100;
	DIR2: BOOL;
	DIR3: BOOL;
	
	car_M1toM2: BOOL;
	motion_flag: BOOL;
	M1toM2_ton: Ton;
	M2Pos2_ftrig: f_trig;
	M1R_Start_rtrig: R_trig;
	car_M2toM1: BOOL;
	M2Pos1_Rtrig: R_TRIG;
	
	car_M2toM3: BOOL;
	car_M3toM2: BOOL;
	M3Pos2_ftrig: F_TRIG;
	M2Pos1_Ftrig: F_TRIG;
	M12: BOOL;
	M21: BOOL;
	M23: BOOL;
	M32: BOOL;
	
	LM_delay: TON;
	LM_delay_trig: R_TRIG;
	LM_Stop_delay: TON;
	LM_Stop_delay_trig: R_TRIG;
	LM_manual_flag: BOOL;
	RM_manual_flag:BOOL;
	RM_delay: TON;
	RM_delay_trig: R_TRIG;
	RM_Stop_delay: TON;
	RM_Stop_delay_trig: R_TRIG;
	LM_Stop_flag: BOOL;
	RM_Stop_flag: BOOL;
	MM1: BOOL;
	MM23: BOOL;
	
	LM_GoLeft:BOOL;
	LM_GoRight:BOOL;
	RM_GoLeft:BOOL;
	RM_GoRight:BOOL;
	LM_Stop:BOOL;
	RM_Stop:BOOL;
	
	MoveVelocity_func: MC_MoveVelocity;
	swinging:BOOL;
	swing_dir: BOOL;
	swing_init:BOOL;
	swing_velocity: UINT:=100;
	swing_interlock:bool;
	stop_swing: BOOL;
	swing_enable:BOOL;
	swing_ton1:TON;
	swing_ton2:TON;
	swing_trig1:R_TRIG;
	swing_trig2:R_TRIG;
	swing_stop_delay:TON;
	swing_stop_trig:R_TRIG;
	swing_start:BOOL;
	swing_stop_Q: BOOL;
	swing_trig2_Q: BOOL;
	swing_ton1_in: BOOL;
	swing_ton2_in: BOOL;
	swing_stop_delay_in: BOOL;
	swing_trig1_Q: BOOL;
	swing_stop_flag: BOOL;
	swing_ton2_PT: TIME:=T#0.8S;
	swing_ton1_PT: TIME:=T#0.2S;
	swing_stop_PT: time:=T#1s;
	swing_stop_flag_time:TON;
	swing_stop_flag_prs:R_TRIG;
	prs_in: BOOL;
	cur_step: INT;
	step1_delay: TON;
	step1_trig: R_TRIG;
	step1_finish: BOOL;
	step2_delay: TON;
	step2_finish: BOOL;
	step2_trig: R_TRIG;
	Rec_MFC1: BOOL;
	Rec_MFC2: BOOL;
	step3_delay: TON;
	step3_finish: BOOL;
	step3_trig: R_TRIG;
	Rec_MFC1_delay: TIME;
	step4_delay: TON;
	step4_trig: R_TRIG;
	step4_finish: BOOL;
	Rec_MFC2_delay: TIME;
	step7_finish: BOOL;
	step7_delay: TON;
	step7_trig: R_TRIG;
	
	M1ToM2_delay: TON;
	M1ToM2_trig: R_TRIG;
	
	ON_POS_delay: TON;
	ON_POS_trig: R_TRIG;
	
	M2ToM3_delay: TON;
	M2ToM3_trig: R_TRIG;
	
	M3ToM2_delay: TON;
	M3ToM2_trig: R_TRIG;
	
	M2ToM1_delay: TON;
	M2ToM1_trig: R_TRIG;
	x: INT;
	swing_Exe: BOOL;
	Rec_finish_trig: R_TRIG;
	Rec_finish_delay: TON;
	Rec_finish_in: BOOL;
	Rec_swing_stop: BOOL;
	Rec_swing_trig: R_TRIG;
	Rec_swing_stop_trig: R_TRIG;
	Rec_swing_reset: BOOL;
	Rec_swing_reset_delay:TON;
END_VAR

manual();	

	IF NOT init THEN
		Pwr_En_1:=1;
		Pwr_En_2:=1;
		Pwr_En_3:=1;
		init:=1;
	END_IF

IF DIR1 THEN
	MoveVelocity_1.Direction:=MC_Positive_Direction;
	ELSE
	MoveVelocity_1.Direction:=MC_Negative_Direction;	
END_IF
IF DIR2 THEN
	MoveVelocity_2.Direction:=MC_Negative_Direction;
	ELSE
	MoveVelocity_2.Direction:=MC_Positive_Direction;	
END_IF

IF DIR3 THEN
	MoveVelocity_3.Direction:=MC_Positive_Direction;
	ELSE
	MoveVelocity_3.Direction:=MC_Negative_Direction;	
END_IF


Power_1(
	Axis:=Axis1 , 
	Enable:= Pwr_En_1, 
	Enable_Positive:=1, 
	Enable_Negative:=1, 
	Override:= 100.0, 
	BufferMode:= , 
	Options:= , 
	Status=> , 
	Busy=> , 
	Active=> , 
	Error=> Pwr1_Err, 
	ErrorID=>Pwr1_ErrId );

MoveStop_1(
	Axis:= Axis1, 
	Execute:= stop_1,
	Deceleration:= Axis1_Speed/10, 
	Jerk:= , 
	Options:= , 
	Done=> , 
	Busy=> , 
	Active=> , 
	CommandAborted=> , 
	Error=> , 
	ErrorID=> );

AxisReset_1(
	Axis:= Axis1, 
	Execute:= reset_1, 
	Done=> , 
	Busy=> , 
	Error=> , 
	ErrorID=> );
	
MoveVelocity_1(
	Axis:= Axis1, 
	Execute:= V_ex1, 
	Velocity:= VV1, 
	Acceleration:= , 
	Deceleration:= , 
	Jerk:= , 
	Direction:= , 
	BufferMode:= , 
	Options:= , 
	InVelocity=> , 
	Busy=> , 
	Active=> , 
	CommandAborted=> , 
	Error=> , 
	ErrorID=> );	
Power_2(
	Axis:=Axis2 , 
	Enable:= Pwr_En_2, 
	Enable_Positive:=1, 
	Enable_Negative:=1, 
	Override:= 100.0, 
	BufferMode:= , 
	Options:= , 
	Status=> , 
	Busy=> , 
	Active=> , 
	Error=> Pwr1_Err, 
	ErrorID=>Pwr1_ErrId );

MoveStop_2(
	Axis:= Axis2, 
	Execute:= stop_2,
	Deceleration:= Axis2_Speed/10, 
	Jerk:= , 
	Options:= , 
	Done=> , 
	Busy=> , 
	Active=> , 
	CommandAborted=> , 
	Error=> , 
	ErrorID=> );

AxisReset_2(
	Axis:= Axis2, 
	Execute:= reset_2, 
	Done=> , 
	Busy=> , 
	Error=> , 
	ErrorID=> );
	
MoveVelocity_2(
	Axis:= Axis2, 
	Execute:= V_ex2, 
	Velocity:= VV2, 
	Acceleration:= , 
	Deceleration:= , 
	Jerk:= , 
	Direction:= , 
	BufferMode:= , 
	Options:= , 
	InVelocity=> , 
	Busy=> , 
	Active=> , 
	CommandAborted=> , 
	Error=> , 
	ErrorID=> );	
	
	Power_3(
	Axis:=Axis3 , 
	Enable:= Pwr_En_3, 
	Enable_Positive:=1, 
	Enable_Negative:=1, 
	Override:= 100.0, 
	BufferMode:= , 
	Options:= , 
	Status=> , 
	Busy=> , 
	Active=> , 
	Error=> Pwr1_Err, 
	ErrorID=>Pwr1_ErrId );

MoveStop_3(
	Axis:= Axis3, 
	Execute:= stop_3,
	Deceleration:= Axis3_Speed/10, 
	Jerk:= , 
	Options:= , 
	Done=> , 
	Busy=> , 
	Active=> , 
	CommandAborted=> , 
	Error=> , 
	ErrorID=> );

AxisReset_3(
	Axis:= Axis3, 
	Execute:= reset_3, 
	Done=> , 
	Busy=> , 
	Error=> , 
	ErrorID=> );
	
MoveVelocity_3(
	Axis:= Axis3, 
	Execute:= V_ex3, 
	Velocity:= VV3, 
	Acceleration:= , 
	Deceleration:= , 
	Jerk:= , 
	Direction:= , 
	BufferMode:= , 
	Options:= , 
	InVelocity=> , 
	Busy=> , 
	Active=> , 
	CommandAborted=> , 
	Error=> , 
	ErrorID=> );

//mainbase button
IF MAIN.M2_SNR1 AND MAIN.M2_SNR2 THEN
	swing_enable:=1;
ELSE
	swing_enable:=0;
END_IF

IF (swinging = 1 AND (swing_enable = 1 OR swing_start = 1)) OR swing_btn THEN
//IF swinging = 1 OR swing_btn = 1 THEN
	Swinging_func();
	swing_start:=1;
	swing_stop_flag:=1;
	prs_in:=0;
ELSE
	IF swing_stop_flag AND prs_in = 0 THEN
		stop_1:=1;
		swing_stop_flag:=0;
		MoveVelocity_func.Execute:=False;
		prs_in:=1;
	END_IF
	swing_start:=0;
	swing_init:=0;
END_IF
swing_stop_flag_time(IN:=prs_in,PT:=T#0.05S,Q=>);
swing_stop_flag_prs(CLK:=swing_stop_flag_time.Q,Q=>);
IF swing_stop_flag_prs.Q THEN
	stop_1:=0;
	stop_swing:=0;
	swing_ton1_in:=0;
	swing_ton2_in:=0;
	swing_Exe:=0;
	swing_stop_delay_in:=0;
END_IF

(*
//Recipe control swinging
IF swing_btn = 1 THEN
	Swinging_func();
	swing_start:=1;
	Rec_swing_stop:=0;
ELSE
	Rec_swing_stop:=1;
END_IF
Rec_swing_stop_trig(CLK:=Rec_swing_stop,Q=>);
IF Rec_swing_stop_trig.Q THEN
	stop_1:=1;
	stop_swing:=1;
	swing_Exe:=0;
	Rec_swing_reset:=1;
END_IF
Rec_swing_reset_delay(IN:=Rec_swing_reset,PT:=T#0.1S,Q=>);
Rec_swing_trig(CLK:=Rec_swing_reset_delay.Q,Q=>);
IF Rec_swing_trig.Q = 1 THEN //常常FASLE
	stop_1:=0;
	stop_swing:=0;
	swing_Exe:=0;
	swing_ton1_in:=0;
	swing_ton2_in:=0;
	swing_stop_delay_in:=0;
	swing_init:=0;
	Rec_swing_reset:=0;
END_IF
*)
Auto();
	

//Motion M1<>M2 M2<>M3
(*  
	IF car_M1toM2 THEN
    stop_1:=0;  
	stop_2:=0;
    stop_3:=0;
	DIR1:=0;
	motion_flag:=1;
	M12:=1;
	END_IF
	
	IF car_M2toM1 THEN
    stop_1:=0;  
	stop_2:=0;
	stop_3:=0;
	DIR1:=1;
	motion_flag:=1;
	M21:=1;
	END_IF

	IF car_M2toM3 THEN
    stop_1:=0;  
	stop_2:=0;
	stop_3:=0;
	DIR1:=0;
	DIR2:=1;
	DIR3:=1;
	motion_flag:=1;
	M23:=1;
	END_IF
	
	IF car_M3toM2 THEN
    stop_1:=0;  
	stop_2:=0;
	stop_3:=0;
	DIR1:=1;
	DIR2:=0;
	DIR3:=0;
	motion_flag:=1;
	M32:=1;
	END_IF

	M1toM2_ton(in:=motion_flag,pt:=T#1S,et=>,q=>);
	M1R_Start_rtrig(CLK:=M1toM2_ton.Q,q=>);
  
	IF M1R_Start_rtrig.Q THEN
		motion_flag:=0;
		IF M32 OR M23 THEN 
		  V_ex1:=1;
		  V_ex2:=1; 
		  V_ex3:=1;
		ELSE
		  V_ex1:=1;
		END_IF	  
	ELSE 
	  V_ex1:=0; 
	  V_ex2:=0; 
	  V_ex3:=0;
	END_IF
  
	IF M12 AND NOT DIR1 THEN
	M2Pos2_ftrig(clk:=di0_2,q=>);
	 IF  M2Pos2_ftrig.Q THEN
	  M12:=0;
	  stop_1:=1;
	 ELSE
	  stop_1:=0;  
	 END_IF 
	END_IF
 
	IF M21 AND DIR1 THEN
	 M2Pos1_Rtrig(clk:=di0_1,q=>);
 	 IF  NOT DI0_0 AND M2Pos1_Rtrig.Q THEN
	 M21:=0;
     stop_1:=1;
	 ELSE
	 stop_1:=0;  
	 END_IF
	END_IF
  
  // M2 TO M3 
  
	IF  M23 AND NOT DIR1 THEN
 		M3Pos2_ftrig(clk:=di0_4,q=>);
		IF M3Pos2_ftrig.Q THEN
			M23:=0;
	 		stop_1:=1;
	    	stop_2:=1;
	    	stop_3:=1;
		ELSE
	 		stop_1:=0;  
	    	stop_2:=0;
	    	stop_3:=0;	
		END_IF
	END_IF
 
	IF M32 AND  DIR1 THEN
		M2Pos1_Ftrig(clk:=di0_1,q=>);
		IF M2Pos1_Ftrig.Q THEN
			M32:=0;
			stop_1:=1;
	   		stop_2:=1;
	    	stop_3:=1;
		ELSE
			stop_1:=0;  
			stop_2:=0;
			stop_3:=0;
		END_IF
	END_IF
  
 *)

ACTION Auto:
//M1 to M2
IF M1ToM2 = 1 THEN
	stop_1:=0;  
	DIR1:=0;
	M1ToM2_flag:=1;
END_IF

//M1ToM2_delay(IN:=M1ToM2_flag,PT:=T#0.1S,Q=>);
//M1ToM2_trig(CLK:=M1ToM2_delay.Q,Q=>);
M1ToM2_trig(CLK:=M1ToM2_flag,Q=>);

IF M1ToM2_trig.Q THEN
	V_ex1:=1;
END_IF

//M2 to M3
IF M2ToM3 = 1 THEN
	stop_1:=0;
	stop_2:=0;
	stop_3:=0;
	V_ex1:=0;
	V_ex2:=0;
	V_ex3:=0;
	DIR1:=0;
	DIR2:=1;
	DIR3:=1;
	M2ToM3_flag:=1;
END_IF

//M2ToM3_delay(IN:=M2ToM3_flag,PT:=T#0.1S,Q=>);
//M2ToM3_trig(CLK:=M2ToM3_delay.Q,Q=>);
M2ToM3_trig(CLK:=M2ToM3_flag,Q=>);

IF M2ToM3_trig.Q THEN
	V_ex1:=1;
	V_ex2:=1;
	V_ex3:=1;
END_IF


//M3 to M2
IF M3ToM2 = 1 THEN
	stop_1:=0;
	stop_2:=0;
	stop_3:=0;
	DIR1:=1;
	DIR2:=0;
	DIR3:=0;
	M3ToM2_flag:=1;
END_IF

//M3ToM2_delay(IN:=M3ToM2_flag,PT:=T#0.1S,Q=>);
//M3ToM2_trig(CLK:=M3ToM2_delay.Q,Q=>);
M3ToM2_trig(CLK:=M3ToM2_flag,Q=>);

IF M3ToM2_trig.Q THEN
	V_ex1:=1;
	V_ex2:=1;
	V_ex3:=1;
END_IF

//M2 to M1
IF M2ToM1 = 1 THEN
	stop_1:=0;  
	DIR1:=1;
	M2ToM1_flag:=1;
END_IF

//M2ToM1_delay(IN:=M2ToM1_flag,PT:=T#0.1S,Q=>);
//M2ToM1_trig(CLK:=M2ToM1_delay.Q,Q=>);
M2ToM1_trig(CLK:=M2ToM1_flag,Q=>);

IF M2ToM1_trig.Q THEN
	V_ex1:=1;
END_IF

IF GVL.ON_POS THEN
	M1ToM2_flag:=0;
	M2ToM3_flag:=0;
	M3ToM2_flag:=0;
	M2ToM1_flag:=0;
	M1ToM2:=0;
	M2ToM3:=0;
	M3ToM2:=0;
	M2ToM1:=0;
	stop_1:=1;
	stop_2:=1;
	stop_3:=1;
	V_ex1:=0;
	V_ex2:=0;
	V_ex3:=0;
	ON_POS_FLAG:=1;
END_IF

//on position and reset
ON_POS_delay(IN:=ON_POS_FLAG,PT:=T#0.1S,Q=>);
ON_POS_trig(CLK:=ON_POS_delay.Q,Q=>);

IF ON_POS_trig.Q THEN
	//ON_POS:=0;
	stop_1:=0;
	stop_2:=0;
	stop_3:=0;
	ON_POS_FLAG:=0;
END_IF

IF Rec_finish THEN
	V_ex1:=0;
	V_ex2:=0;
	V_ex3:=0;
	Rec_finish_in:=1;
	stop_1:=1;
	stop_2:=1;
	stop_3:=1;
END_IF
Rec_finish_delay(IN:=Rec_finish_in,PT:=T#0.2S,Q=>);
Rec_finish_trig(CLK:=Rec_finish_delay.Q,Q=>);
IF Rec_finish_trig.Q THEN
	Rec_finish_in:=0;
	stop_1:=0;
	stop_2:=0;
	stop_3:=0;
END_IF
END_ACTION

ACTION manual:
//M1 --> M2
IF LM_GoRight = 1 AND MM1 = 0 THEN
	stop_1:=0;  
	DIR1:=0;
	Lm_manual_flag:=1;
	MM1:=1;
END_IF
//M2 --> M1
IF LM_GoLeft = 1 AND MM1 = 0 THEN
	stop_1:=0;  
	DIR1:=1;
	Lm_manual_flag:=1;
	MM1:=1;
END_IF

LM_delay(IN:=Lm_manual_flag,PT:=T#0.1S,Q=>);
LM_delay_trig(CLK:=LM_delay.Q,Q=>);

IF LM_delay_trig.Q THEN
	Lm_manual_flag:=0;
	V_ex1:=1;
END_IF

//LM stop

IF LM_Stop = 1 AND MM1 = 1 THEN
	LM_GoLeft:=0;
	LM_GoRight:=0;
	LM_Stop_flag:=1;
END_IF

LM_Stop_delay(IN:=LM_Stop_flag,PT:=T#0.1S,Q=>);
LM_Stop_delay_trig(CLK:=LM_Stop_delay.Q,Q=>);

IF LM_Stop_delay_trig.Q = 1 THEN
	LM_Stop_flag:=0;
	V_ex1:=0;
	stop_1:=1;
	MM1:=0;
END_IF

//#####################################

//M2 --> M3
IF RM_GoRight = 1 AND MM23 = 0 THEN
	stop_2:=0;
	stop_3:=0;
	DIR2:=1;
	DIR3:=1;
	Rm_manual_flag:=1;
	MM23 := 1;
END_IF
//M3 --> M2
IF RM_GoLeft = 1 AND MM23 = 0  THEN
	stop_2:=0;
	stop_3:=0;
	DIR2:=0;
	DIR3:=0;
	Rm_manual_flag:=1;
	MM23 := 1;
END_IF

RM_delay(IN:=Rm_manual_flag,PT:=T#0.1S,Q=>);
RM_delay_trig(CLK:=RM_delay.Q,Q=>);

IF RM_delay_trig.Q THEN
	Rm_manual_flag:=0;
	V_ex2:=1;
	V_ex3:=1;
END_IF

//RM stop
IF RM_Stop = 1 AND MM23 = 1 THEN
	RM_GoRight:=0;
	RM_GoLeft:=0;
	RM_Stop_flag:=1;
END_IF

RM_Stop_delay(IN:=RM_Stop_flag,PT:=T#0.1S,Q=>);
RM_Stop_delay_trig(CLK:=RM_Stop_delay.Q,Q=>);


IF RM_Stop_delay_trig.Q = 1 THEN
	RM_Stop_flag:=0;
	V_ex2:=0;
	V_ex3:=0;
	stop_2:=1;
	stop_3:=1;
	MM23:=0;
END_IF
END_ACTION

ACTION Swinging_func:
MoveVelocity_func(
	Axis:= Axis1, 
	Execute:= swing_Exe, 
	Velocity:= swing_velocity, 
	Acceleration:= , 
	Deceleration:= , 
	Jerk:= , 
	Direction:= , 
	BufferMode:= , 
	Options:= , 
	InVelocity=> , 
	Busy=> , 
	Active=> , 
	CommandAborted=> , 
	Error=> , 
	ErrorID=> );
	
MoveStop_1(
	Axis:= Axis1, 
	Execute:= stop_swing,
	Deceleration:= Axis1_Speed/10, 
	Jerk:= , 
	Options:= , 
	Done=> , 
	Busy=> , 
	Active=> , 
	CommandAborted=> , 
	Error=> , 
	ErrorID=> );

IF NOT swing_init THEN
	MoveVelocity_func.Direction:=mc_positive_direction;// go right
	swing_Exe:=TRUE;
	swing_ton1_in:=TRUE;
	swing_init:=1;
	swing_dir:=1;
END_IF

swing_ton1(IN:=swing_ton1_in,PT:=swing_ton1_PT,Q=>);
swing_ton2(IN:=swing_ton2_in,PT:=swing_ton2_PT,Q=>);
swing_trig1(CLK:=swing_ton1.Q,Q=>swing_trig1_Q);
swing_trig2(CLK:=swing_ton2.Q,Q=>swing_trig2_Q);
swing_stop_delay(IN:=swing_stop_delay_in,PT:=swing_stop_PT,Q=>);
swing_stop_trig(CLK:=swing_stop_delay.Q,Q=>swing_stop_Q);

IF swing_trig1_Q = 1 THEN
	swing_ton1_in:=FALSE;
	stop_swing:=1;
	swing_Exe:=FALSE;
	swing_stop_delay_in:=TRUE;
END_IF

IF swing_stop_Q AND swing_init = 1 THEN
	swing_dir:=NOT swing_dir;
	IF swing_dir = 0 THEN
		MoveVelocity_func.Direction:=mc_negative_direction;
	ELSE
		MoveVelocity_func.Direction:=mc_positive_direction;
	END_IF
	swing_stop_delay_in:=FALSE;
	stop_swing:=0;
	swing_ton2_in:=TRUE;
	swing_Exe:=TRUE;
END_IF

IF swing_trig2_Q THEN
	stop_swing:=1;
	swing_ton2_in:=FALSE;
	swing_Exe:=FALSE;
	swing_stop_delay_in:=TRUE;
END_IF
END_ACTION

END_PROGRAM

// ---- GlobalTextList.TcGTLO
TEXTLIST GlobalTextList
  567 = '\n'
  747 = '$d'
  397 = '%'
  290 = '%.2f'
  172 = '%3.1f'
  449 = '%3.2f'
  91 = '%4.1f'
  77 = '%b'
  742 = '%c'
  304 = '%D'
  600 = '%d'
  1523 = '%f'
  209 = '%s'
  1444 = '(%)'
  360 = '(porr)'
  1013 = '(torr)'
  903 = '123'
  1416 = '3L_Cyn1_Shr\n'
  511 = 'ALARM'
  341 = 'ATM1'
  447 = 'ATM2'
  611 = 'ATM3'
  108 = 'Axis 1'
  853 = 'AXIS1'
  289 = 'AXIS2'
  786 = 'AXIS3'
  131 = 'BG1'
  773 = 'Buzzer'
  598 = 'Buzzer\n'
  712 = 'CG1'
  328 = 'CG2'
  653 = 'CG3'
  329 = 'Clear'
  426 = 'close'
  702 = 'CLOSE'
  1763 = 'Copy last recipe'
  851 = 'Copy last step'
  1664 = 'Delay'
  435 = 'DIR'
  1270 = 'Down'
  973 = 'DOWN'
  1773 = 'Edit'
  229 = 'Execute'
  194 = 'EXH'
  995 = 'EXHAST'
  1574 = 'GAS inlet Pressure'
  375 = 'Gas Inlet Pressure'
  465 = 'GASnlet Pressure'
  64 = 'GGG'
  915 = 'GGGGG'
  632 = 'Green'
  249 = 'Green\n'
  1020 = 'GSnlet Pressure'
  138 = 'GV1'
  720 = 'GV1 SENEOR'
  862 = 'GV1_Cyn_Ext'
  402 = 'GV1_Cyn_Ext\n'
  835 = 'GV1_Cyn_Ext_Snr\n'
  1509 = 'GV1_Cyn_Shr'
  847 = 'GV1_Cyn_Shr\n'
  955 = 'GV1_Cyn_Shr_Snr\n'
  948 = 'GV1_Ext_Snr\n'
  193 = 'GV1_Shr_Snr\n'
  396 = 'GV2'
  605 = 'GV2 SENSOR'
  1 = 'GV2_Cyn_Ext'
  666 = 'GV2_Cyn_Ext\n'
  631 = 'GV2_Cyn_Ext_Snr\n'
  729 = 'GV2_Cyn_Shr\n'
  910 = 'GV2_Cyn_Shr_Snr\n'
  1341 = 'GV2_Ext_Snr\n'
  21 = 'GV2_Shr_Snr\n'
  388 = 'H1'
  574 = 'H2'
  1101 = 'HEATER COOLING'
  1561 = 'heater Settining'
  1056 = 'heater Temp Settining'
  216 = 'HEATER1 TEMP'
  1367 = 'HEATER1 TEMPrs'
  1566 = 'HEATER2 TEMP'
  601 = 'HTC Set Position'
  1082 = 'IN'
  710 = 'Insert'
  986 = 'IO'
  2145 = 'KPA'
  507 = 'LV80'
  983 = 'LV80 SW85\n'
  122 = 'LV80 SW90\n'
  373 = 'LV80 SW_85\n'
  63 = 'LV80 SW_90\n'
  800 = 'LV80 Trip\n'
  530 = 'M1'
  238 = 'M1 (Roller)'
  223 = 'M1 Roller'
  904 = 'M1 to M2'
  947 = 'M2'
  533 = 'M2 (MA)'
  119 = 'M2 Pressure Settining'
  2131 = 'M2 to M1'
  2290 = 'M2 to M3'
  319 = 'M3'
  97 = 'M3 (HEATER)'
  688 = 'M3 Pressure Settining'
  1440 = 'M3 to M2'
  6 = 'M3L_Cyn1_Ext'
  506 = 'M3L_Cyn1_Ext\n'
  827 = 'M3L_Cyn1_Ext_Snr\n'
  100 = 'M3L_Cyn1_Shr'
  287 = 'M3L_Cyn1_Shr\n'
  789 = 'M3L_Cyn1_Shr_Snr\n'
  1017 = 'M3L_Cyn2_Ext'
  527 = 'M3L_Cyn2_Ext\n'
  750 = 'M3L_Cyn2_Ext_Snr'
  214 = 'M3L_Cyn2_Shr\n'
  5 = 'M3L_Cyn2_Shr_Snr\n'
  481 = 'M3R_Cyn1_Ext'
  861 = 'M3R_Cyn1_Ext\n'
  949 = 'M3R_Cyn1_Ext_Snr'
  1313 = 'M3R_Cyn1_Shr'
  479 = 'M3R_Cyn1_Shr\n'
  1205 = 'M3R_Cyn1_Shr\n\n'
  58 = 'M3R_Cyn1_Shr\nM3R_Cyn1_Shr\n'
  137 = 'M3R_Cyn1_Shr_Snr\n'
  318 = 'M3R_Cyn2_Ext\n'
  890 = 'M3R_Cyn2_Ext_Snr\n'
  81 = 'M3R_Cyn2_Shr\n'
  458 = 'M3R_Cyn2_Shr_Snr\n'
  274 = 'M3V_Cyn1_Ext'
  496 = 'M3V_Cyn1_Ext\n'
  368 = 'M3V_Cyn1_Ext_Snr\n'
  239 = 'M3V_Cyn1_Shr'
  546 = 'M3V_Cyn1_Shr\n'
  776 = 'M3V_Cyn1_Shr_Snr\n'
  1231 = 'MAIN'
  38 = 'MA_SOURCE'
  1256 = 'MA_SRY'
  1023 = 'MFC1'
  1306 = 'MFC1 button'
  1419 = 'MFC1 Button'
  767 = 'MFC1 DEV'
  23 = 'MFC1 Setting'
  390 = 'MFC1 SP'
  36 = 'MFC2'
  572 = 'MFC2 Button'
  1192 = 'MFC2 DEV'
  939 = 'MFC2 Setting'
  571 = 'MFC2 SP'
  1288 = 'MOTION'
  377 = 'N2'
  503 = 'NC1'
  647 = 'NC10'
  599 = 'NC11'
  0 = 'NC12'
  957 = 'NC13'
  517 = 'NC14'
  37 = 'NC2'
  392 = 'NC23'
  737 = 'NC3'
  976 = 'NC4'
  170 = 'NC5'
  542 = 'NC6'
  140 = 'NC7'
  400 = 'NC8'
  338 = 'NC9'
  686 = 'NH3'
  1100 = 'open'
  885 = 'OPEN'
  703 = 'OUT'
  147 = 'PARAMETER'
  482 = 'Position Setting'
  570 = 'Pos_M1_1\n'
  34 = 'Pos_M2_1\n'
  96 = 'Pos_M2_2\n'
  389 = 'Pos_M3_1\n'
  468 = 'Pos_M3_2\n'
  215 = 'Pos_M3_3\n'
  543 = 'Pos_Snr_M1_1\n'
  353 = 'Pos_Snr_M1_1\n(PSI)'
  90 = 'Pos_Snr_M2_1\n'
  452 = 'Pos_Snr_M2_2\n'
  597 = 'Pos_Snr_M3_1\n'
  749 = 'Pos_Snr_M3_2\n'
  25 = 'Pos_Snr_M3_3\n'
  648 = 'Pr Mode'
  608 = 'Pressure 1(PSI)'
  306 = 'Prs_In'
  1333 = 'psi'
  654 = 'PUMP COOLING'
  1799 = 'PUT DOWN'
  448 = 'Put down'
  2426 = 'Rec Cancel'
  2205 = 'Rec Init'
  1498 = 'Rec Start'
  1826 = 'Rec Stop'
  961 = 'Recipe'
  554 = 'Recipe Name'
  2199 = 'Recipt'
  743 = 'Recipt Name'
  854 = 'Red\n'
  777 = 'RESET'
  1218 = 'reset'
  51 = 'RESSET'
  429 = 'RV1'
  614 = 'RV2'
  2537 = 'Save'
  393 = 'sccm'
  480 = 'SERVER ON'
  765 = 'Set to Position'
  171 = 'slm'
  433 = 'SPEED'
  518 = 'Start'
  1705 = 'Step 1'
  104 = 'Step 10'
  544 = 'Step 13'
  1246 = 'Step 2'
  2038 = 'Step 3'
  1131 = 'Step 4'
  1891 = 'Step 5'
  1039 = 'Step 6'
  196 = 'Step 7'
  708 = 'Step 8'
  1268 = 'Step 9'
  934 = 'Step Name'
  312 = 'STOP'
  1543 = 'SV1'
  113 = 'SV2'
  1656 = 'SV3'
  219 = 'Swing'
  1018 = 'Swinging'
  836 = 'TAKE UP'
  2538 = 'Take up'
  526 = 'Time (Sec)'
  636 = 'torr'
  288 = 'TV'
  545 = 'up'
  1906 = 'UP'
  48 = 'VB1'
  55 = 'VB1\n'
  671 = 'VB12'
  738 = 'VB13'
  485 = 'VB2'
  453 = 'VB3'
  758 = 'VB4'
  454 = 'VEN3'
  175 = 'VEN32'
  804 = 'VENT1'
  806 = 'Vent1'
  646 = 'Vent1\n'
  850 = 'Vent12'
  692 = 'Vent13'
  881 = 'Vent2'
  128 = 'VENT2'
  604 = 'Vent3'
  430 = 'VENT3'
  790 = 'WATER Prs'
  1863 = 'WATER TEMP'
  1362 = 'WaterFlow_SW1\n'
  825 = 'WaterFlow_SW2'
  106 = 'WaterFlow_SW3'
  124 = 'Water_Flow_SW1\n'
  395 = 'Water_Flow_SW13'
  829 = 'Water_Flow_SW2'
  535 = 'Water_Flow_SW3'
  1099 = 'WSU251'
  188 = 'WSU251\n'
  405 = 'WSU251 Trip\n'
  590 = 'WSU251\u3000\n'
  1380 = 'WtrFlow_SW1\n'
  534 = 'WtrFlow_SW2'
  372 = 'WtrFlow_SW3'
  502 = 'Wtr_Flow_SW1\n'
  1295 = 'Yellow'
  132 = 'Yellow\n'
END_TEXTLIST

// ---- Recipt_no.TcTLO
TEXTLIST Recipt_no
  1 = 'Recipe 1'
  2 = 'Recipe 2'
  3 = 'Recipe 3'
  4 = 'Recipe 4'
  5 = 'Recipe 5'
  6 = 'Recipe 6'
  7 = 'Recipe 7'
  8 = 'Recipe 8'
  9 = 'Recipe 9'
  10 = 'Recipe 10'
   = ''
END_TEXTLIST

// ---- step.TcTLO
TEXTLIST step
  1 = 'Step 1'
  2 = 'Step 2'
  3 = 'Step 3'
  4 = 'Step 4'
  5 = 'Step 5'
  6 = 'Step 6'
  7 = 'Step 7'
  8 = 'Step 8'
  9 = 'Step 9'
  10 = 'Step 10'
  11 = 'Step 11'
  12 = 'Step 12'
  13 = 'Step 13'
  14 = 'Step 14'
  15 = 'Step 15'
  16 = 'Step 16'
  17 = 'Step 17'
  18 = 'Step 18'
  19 = 'Step 19'
  20 = 'Step 20'
  21 = 'Step 21'
  22 = 'Step 22'
  23 = 'Step 23'
  24 = 'Step 24'
  25 = 'Step 25'
  26 = 'Step 26'
  27 = 'Step 27'
  28 = 'Step 28'
  29 = 'Step 29'
  30 = 'Step 30'
   = ''
END_TEXTLIST

// ---- VISUs/ALARM.TcVIS
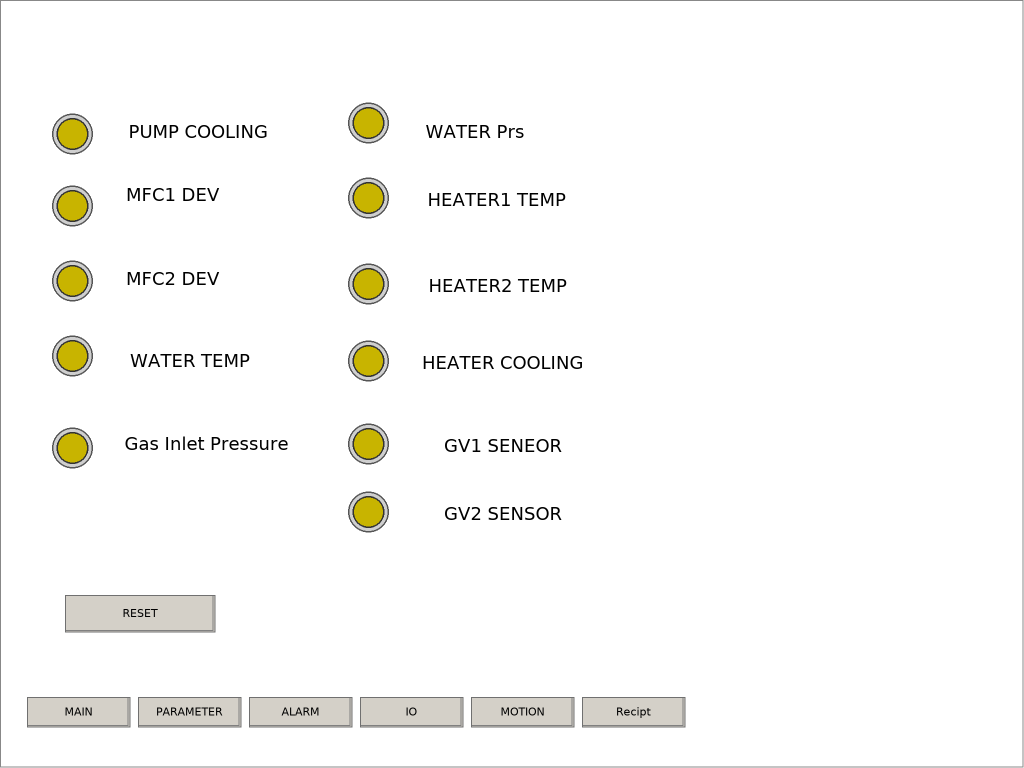
VISUALIZATION ALARM  // 1024x768, background image ImagePool_Base.base
    Button (27,697 103x30), "MAIN"
        OnMouseClick: change screen: MainBase
    Button (138,697 103x30), "PARAMETER"
        OnMouseClick: change screen: PARAMETER
    Button (249,697 103x30), "ALARM"
        OnMouseClick: change screen: ALARM
    Button (360,697 103x30), "IO"
        OnMouseClick: change screen: IO_TABLE
    Button (471,697 103x30), "MOTION"
        OnMouseClick: change screen: MOTION
    Lamp1 (49,109 47x50), variable: MAIN.ALM_PUMP_COOL, style: Lamp-Lamp1-Yellow
    Label (105,117 187x30), "PUMP COOLING"
    Label (116,180 114x30), "MFC1 DEV"
    Label (116,264 114x30), "MFC2 DEV"
    Label (117,346 146x30), "WATER TEMP"
    Label (418,117 114x30), "WATER Prs"
    Lamp1 (49,181 47x50), variable: MAIN.ALM_MFC1_DEV, style: Lamp-Lamp1-Yellow
    Lamp1 (49,256 47x50), variable: MAIN.ALM_MFC2_DEV, style: Lamp-Lamp1-Yellow
    Lamp1 (49,331 47x50), variable: MAIN.ALM_WATER_TEMP, style: Lamp-Lamp1-Yellow
    Lamp1 (345,98 47x50), variable: MAIN.ALM_WATER_Prs, style: Lamp-Lamp1-Yellow
    Lamp1 (345,173 47x50), variable: MAIN.ALM_Heater1_Temp, style: Lamp-Lamp1-Yellow
    Label (395,185 204x30), "HEATER1 TEMP"
    Lamp1 (345,259 47x50), variable: MAIN.ALM_Heater2_Temp, style: Lamp-Lamp1-Yellow
    Label (396,271 204x30), "HEATER2 TEMP"
    Lamp1 (345,336 47x50), variable: MAIN.ALM_Heater_cool, style: Lamp-Lamp1-Yellow
    Label (401,348 204x30), "HEATER COOLING"
    Lamp1 (49,423 47x50), variable: MAIN.ALM_inlet_prs, style: Lamp-Lamp1-Yellow
    Label (111,429 191x30), "Gas Inlet Pressure"
    Lamp1 (345,419 47x50), variable: MAIN.ALM_GV1_Snr, style: Lamp-Lamp1-Yellow
    Label (401,431 204x30), "GV1 SENEOR"
    Lamp1 (345,487 47x50), variable: MAIN.ALM_GV2_Snr, style: Lamp-Lamp1-Yellow
    Label (401,499 204x30), "GV2 SENSOR"
    Button (65,595 150x37), "RESET"
        tap MAIN.RST_BTN p1329445385=TRUE
    Button (582,697 103x30), "Recipt"
        OnMouseClick: change screen: Recipt
END_VISUALIZATION

// ---- VISUs/IO_TABLE.TcVIS
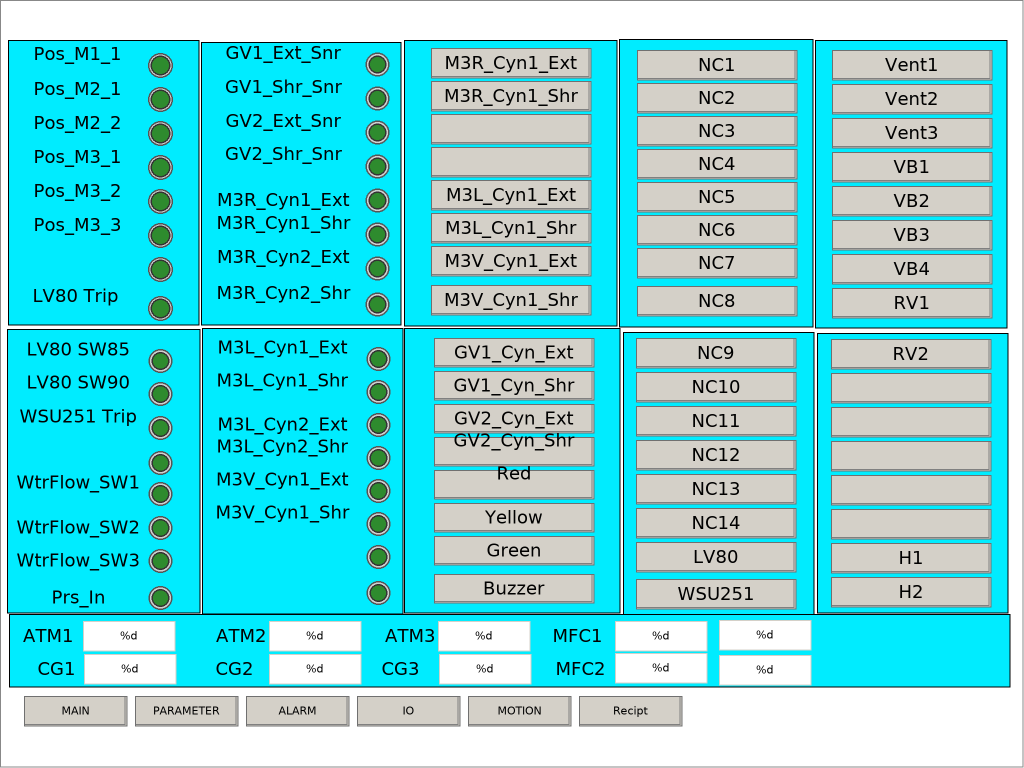
VISUALIZATION IO_TABLE  // 1024x768, background image ImagePool_Base.base
    RoundedRectangle (623,332 191x283)
    RoundedRectangle (619,39 194x288)
    RoundedRectangle (817,333 191x280)
    RoundedRectangle (8,40 191x285)
    Lamp1 (146,83 29x33), variable: DI0_1, style: Lamp-Lamp1-Green
    Lamp1 (146,117 29x33), variable: DI0_2, style: Lamp-Lamp1-Green
    Lamp1 (146,49 29x33), variable: DI0_0, style: Lamp-Lamp1-Green
    Lamp1 (146,185 29x33), variable: DI0_4, style: Lamp-Lamp1-Green
    Lamp1 (146,151 29x33), variable: DI0_3, style: Lamp-Lamp1-Green
    Lamp1 (146,292 29x33), variable: DI0_7, style: Lamp-Lamp1-Green
    Lamp1 (146,253 29x33), variable: DI0_6, style: Lamp-Lamp1-Green
    Lamp1 (146,219 29x33), variable: DI0_5, style: Lamp-Lamp1-Green
    Label (-9,50 173x30), "Pos_M1_1"
    Label (-9,85 173x30), "Pos_M2_1"
    Label (-9,119 173x30), "Pos_M2_2"
    Label (-9,153 173x30), "Pos_M3_1"
    Label (-9,187 173x30), "Pos_M3_2"
    Label (-9,221 173x30), "Pos_M3_3"
    Label (-9,255 173x30)
    Label (-11,292 173x30), "LV80 Trip"
    RoundedRectangle (7,329 193x284)
    Lamp1 (147,378 27x32), variable: DI1_1, style: Lamp-Lamp1-Green
    Lamp1 (147,412 27x32), variable: DI1_2, style: Lamp-Lamp1-Green
    Lamp1 (147,345 27x32), variable: DI1_0, style: Lamp-Lamp1-Green
    Lamp1 (147,478 27x32), variable: DI1_4, style: Lamp-Lamp1-Green
    Lamp1 (147,447 27x32), variable: DI1_3, style: Lamp-Lamp1-Green
    Lamp1 (147,582 27x32), variable: DI1_7, style: Lamp-Lamp1-Green
    Lamp1 (147,545 27x32), variable: DI1_6, style: Lamp-Lamp1-Green
    Lamp1 (147,512 27x32), variable: DI1_5, style: Lamp-Lamp1-Green
    Label (-2,346 161x29), "LV80 SW85"
    Label (-2,379 161x29), "LV80 SW90"
    Label (-2,413 161x29), "WSU251 Trip"
    Label (-2,443 161x29)
    Label (-2,479 161x29), "WtrFlow_SW1"
    Label (-2,513 161x29), "WtrFlow_SW2"
    Label (-2,546 161x29), "WtrFlow_SW3"
    Label (-2,583 161x29), "Prs_In"
    RoundedRectangle (815,40 192x288)
    RoundedRectangle (9,614 1001x73)
    RoundedRectangle (201,42 200x283)
    Lamp1 (364,82 27x33), variable: DI2_1, style: Lamp-Lamp1-Green
    Lamp1 (364,116 27x33), variable: DI2_2, style: Lamp-Lamp1-Green
    Lamp1 (364,48 27x33), variable: DI2_0, style: Lamp-Lamp1-Green
    Lamp1 (364,184 27x33), variable: DI2_4, style: Lamp-Lamp1-Green
    Lamp1 (364,150 27x33), variable: DI2_3, style: Lamp-Lamp1-Green
    Lamp1 (364,252 27x33), variable: DI2_6, style: Lamp-Lamp1-Green
    Lamp1 (364,218 27x33), variable: DI2_5, style: Lamp-Lamp1-Green
    Lamp1 (364,288 27x33), variable: DI2_7, style: Lamp-Lamp1-Green
    Label (196,49 175x30), "GV1_Ext_Snr"
    Label (196,83 175x30), "GV1_Shr_Snr"
    Label (196,117 175x30), "GV2_Ext_Snr"
    Label (196,150 175x30), "GV2_Shr_Snr"
    Label (196,185 175x30), "M3R_Cyn1_Ext"
    Label (196,219 175x30), "M3R_Cyn1_Shr"
    Label (196,253 175x30), "M3R_Cyn2_Ext"
    Label (196,289 175x30), "M3R_Cyn2_Shr"
    RoundedRectangle (202,328 201x286)
    Lamp1 (365,376 27x32), variable: DI3_1, style: Lamp-Lamp1-Green
    Lamp1 (365,409 27x32), variable: DI3_2, style: Lamp-Lamp1-Green
    Lamp1 (365,343 27x32), variable: DI3_0, style: Lamp-Lamp1-Green
    Lamp1 (365,475 27x32), variable: DI3_4, style: Lamp-Lamp1-Green
    Lamp1 (365,442 27x32), variable: DI3_3, style: Lamp-Lamp1-Green
    Lamp1 (365,541 27x32), variable: DI3_6, style: Lamp-Lamp1-Green
    Lamp1 (365,508 27x32), variable: DI3_5, style: Lamp-Lamp1-Green
    Lamp1 (365,577 27x32), variable: DI3_7, style: Lamp-Lamp1-Green
    Label (195,344 175x29), "M3L_Cyn1_Ext"
    Label (195,377 175x29), "M3L_Cyn1_Shr"
    Label (195,410 175x29), "M3L_Cyn2_Ext"
    Label (195,443 175x29), "M3L_Cyn2_Shr"
    Label (195,476 175x29), "M3V_Cyn1_Ext"
    Label (195,509 175x29), "M3V_Cyn1_Shr"
    RoundedRectangle (404,40 213x286)
    Button (431,48 160x30), "M3R_Cyn1_Ext"
        toggle DO0_0
    Button (431,81 160x30), "M3R_Cyn1_Shr"
        toggle DO0_1
    Button (431,114 160x30)
        toggle DO0_2
    Button (431,147 160x30)
        toggle DO0_3
    Button (431,180 160x30), "M3L_Cyn1_Ext"
        toggle DO0_4
    Button (431,213 160x30), "M3L_Cyn1_Shr"
        toggle DO0_5
    Button (431,246 160x30), "M3V_Cyn1_Ext"
        toggle DO0_6
    Button (431,285 160x30), "M3V_Cyn1_Shr"
        toggle DO0_7
    RoundedRectangle (404,328 216x285)
    Button (434,338 160x29), "GV1_Cyn_Ext"
        toggle DO1_0
    Button (434,371 160x29), "GV1_Cyn_Shr"
        toggle DO1_1
    Button (434,404 160x29), "GV2_Cyn_Ext"
        toggle DO1_2
    Button (434,437 160x29), "GV2_Cyn_Shr"
        toggle DO1_3
    Button (434,470 160x29), "Red"
        toggle DO1_4
    Button (434,503 160x29), "Yellow"
        toggle DO1_5
    Button (434,536 160x29), "Green"
        toggle DO1_6
    Button (434,574 160x29), "Buzzer"
        toggle DO1_7
    Button (637,50 160x30), "NC1"
        toggle DO2_0
    Button (637,83 160x30), "NC2"
        toggle DO2_1
    Button (637,116 160x30), "NC3"
        toggle DO2_2
    Button (637,149 160x30), "NC4"
        toggle DO2_3
    Button (637,182 160x30), "NC5"
        toggle DO2_4
    Button (637,215 160x30), "NC6"
        toggle DO2_5
    Button (637,248 160x30), "NC7"
        toggle DO2_6
    Button (637,286 160x30), "NC8"
        toggle DO2_7
    Button (636,338 160x30), "NC9"
        toggle DO3_0
    Button (636,372 160x30), "NC10"
        toggle DO3_1
    Button (636,406 160x30), "NC11"
        toggle DO3_2
    Button (636,440 160x30), "NC12"
        toggle DO3_3
    Button (636,474 160x30), "NC13"
        toggle DO3_4
    Button (636,508 160x30), "NC14"
        toggle DO3_5
    Button (636,542 160x30), "LV80"
        toggle DO3_6
    Button (636,579 160x30), "WSU251"
        toggle DO3_7
    Button (832,50 160x30), "Vent1"
        toggle DO4_0
    Button (832,84 160x30), "Vent2"
        toggle DO4_1
    Button (832,118 160x30), "Vent3"
        toggle DO4_2
    Button (832,152 160x30), "VB1"
        toggle DO4_3
    Button (832,186 160x30), "VB2"
        toggle DO4_4
    Button (832,220 160x30), "VB3"
        toggle DO4_5
    Button (832,254 160x30), "VB4"
        toggle DO4_6
    Button (832,288 160x30), "RV1"
        toggle DO4_7
    Button (831,339 160x30), "RV2"
        toggle DO5_0
    Button (831,373 160x30)
        toggle DO5_1
    Button (831,407 160x30)
        toggle DO5_2
    Button (831,441 160x30)
        toggle DO5_3
    Button (831,475 160x30)
        toggle DO5_4
    Button (831,509 160x30)
        toggle DO5_5
    Button (831,543 160x30), "H1"
        toggle DO5_6
    Button (831,577 160x30), "H2"
        toggle DO5_7
    Label (821,398 161x30)
    Label (821,432 161x30)
    Label (821,466 161x30)
    Label (821,500 161x30)
    Label (821,534 161x30)
    Textfield (83,621 92x30), "%d", text variable: AI0_0
        OnMouseClick: write the text variable via Default, min 0, max 300
    Textfield (269,621 92x30), "%d", text variable: AI0_1
        OnMouseClick: write the text variable via Default, min 0, max 300
    Textfield (438,621 92x30), "%d", text variable: AI0_2
        OnMouseClick: write the text variable via Default, min 0, max 300
    Textfield (84,654 92x30), "%d", text variable: AI0_3
        OnMouseClick: write the text variable via Default, min 0, max 300
    Textfield (269,654 92x30), "%d", text variable: AI1_0
        OnMouseClick: write the text variable via Default, min 0, max 300
    Textfield (439,654 92x30), "%d", text variable: AI1_1
        OnMouseClick: write the text variable via Default, min 0, max 300
    Textfield (615,621 92x30), "%d", text variable: AI1_2
    Textfield (615,653 92x30), "%d", text variable: AI1_3
    Label (21,621 55x30), "ATM1"
    Label (214,621 55x30), "ATM2"
    Label (383,621 55x30), "ATM3"
    Label (29,654 55x30), "CG1"
    Label (207,654 55x30), "CG2"
    Label (373,654 55x30), "CG3"
    Label (550,621 55x30), "MFC1"
    Label (553,654 55x30), "MFC2"
    Textfield (719,620 92x30), "%d", text variable: AO0_2
        OnMouseClick: write the text variable via Default, min 0, max 300
    Textfield (719,655 92x30), "%d", text variable: AO0_3
        OnMouseClick: write the text variable via Default, min 0, max 300
    Button (24,696 103x30), "MAIN"
        OnMouseClick: change screen: MainBase
    Button (135,696 103x30), "PARAMETER"
        OnMouseClick: change screen: PARAMETER
    Button (246,696 103x30), "ALARM"
        OnMouseClick: change screen: ALARM
    Button (357,696 103x30), "IO"
        OnMouseClick: change screen: IO_TABLE
    Button (468,696 103x30), "MOTION"
        OnMouseClick: change screen: MOTION
    Button (579,696 103x30), "Recipt"
        OnMouseClick: change screen: Recipt
END_VISUALIZATION

// ---- VISUs/MainBase.TcVIS
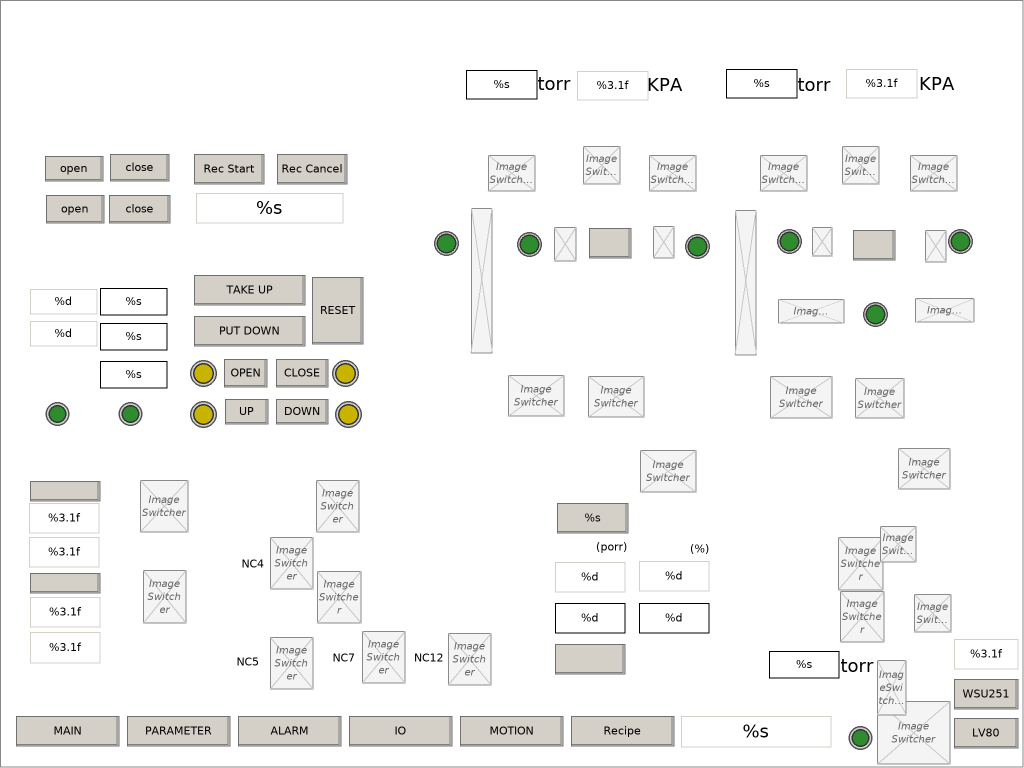
VISUALIZATION MainBase  // 1024x768, background image ImagePool_Base.LAYOUT
    ImageSwitcher (140,480 48x52), variable: DO2_0, background image: ImagePool_Base.VAL_ON, image: ImagePool_Base.VAL_OFF, behaviour: TOGGLE
    ImageSwitcher (143,570 43x53), variable: DO2_1, background image: ImagePool_Base.VAL_ON, image: ImagePool_Base.VAL_OFF, behaviour: TOGGLE
    ImageSwitcher (316,480 43x52), variable: DO2_2, background image: ImagePool_Base.VAL_ON, image: ImagePool_Base.VAL_OFF, behaviour: TOGGLE
    ImageSwitcher (317,571 44x52), variable: DO2_5, background image: ImagePool_Base.VAL_ON, image: ImagePool_Base.VAL_OFF, behaviour: TOGGLE
    ImageSwitcher (838,537 45x53), variable: DO4_0, background image: ImagePool_Base.VAL_ON, image: ImagePool_Base.VAL_OFF, behaviour: TOGGLE
    ImageSwitcher (649,155 47x36), variable: DO4_1, background image: ImagePool_Base.VAL_ON_RL, image: ImagePool_Base.VAL_OFF_RL, behaviour: TOGGLE
    ImageSwitcher (910,155 47x36), variable: DO4_2, background image: ImagePool_Base.VAL_ON_RL, image: ImagePool_Base.VAL_OFF_RL, behaviour: TOGGLE
    ImageSwitcher (840,591 44x51), variable: DO4_3, background image: ImagePool_Base.VAL_ON, image: ImagePool_Base.VAL_OFF, behaviour: TOGGLE
    ImageSwitcher (488,155 47x36), variable: DO4_4, background image: ImagePool_Base.VAL_ON_RL, image: ImagePool_Base.VAL_OFF_RL, behaviour: TOGGLE
    ImageSwitcher (760,155 47x36), variable: DO4_5, background image: ImagePool_Base.VAL_ON_RL, image: ImagePool_Base.VAL_OFF_RL, behaviour: TOGGLE
    ImageSwitcher (588,376 56x41), variable: DO2_7, background image: ImagePool_Base.VAL_ON_RL, image: ImagePool_Base.VAL_OFF_RL, behaviour: TOGGLE
    ImageSwitcher (508,375 56x41), variable: DO3_0, background image: ImagePool_Base.VAL_ON_RL, image: ImagePool_Base.VAL_OFF_RL, behaviour: TOGGLE
    ImageSwitcher (855,378 49x40), variable: DO3_1, background image: ImagePool_Base.VAL_ON_RL, image: ImagePool_Base.VAL_OFF_RL, behaviour: TOGGLE
    ImageSwitcher (770,376 62x42), variable: DO3_2, background image: ImagePool_Base.VAL_ON_RL, image: ImagePool_Base.VAL_OFF_RL, behaviour: TOGGLE
    ImageSwitcher (640,450 56x42), variable: DO4_7, background image: ImagePool_Base.VAL_ON_RL, image: ImagePool_Base.VAL_OFF_RL, behaviour: TOGGLE
    ImageSwitcher (898,448 52x41), variable: DO5_0, background image: ImagePool_Base.VAL_ON_RL, image: ImagePool_Base.VAL_OFF_RL, behaviour: TOGGLE
    ImageSwitcher (778,299 66x24), variable: DO5_6, background image: ImagePool_Base.HTR_ON, image: ImagePool_Base.HTR_OFF, behaviour: TOGGLE
    ImageSwitcher (915,298 59x24), variable: DO5_7, background image: ImagePool_Base.HTR_ON, image: ImagePool_Base.HTR_OFF, behaviour: TOGGLE
    Lamp1 (515,228 29x33), variable: MAIN.M2_SNR1, style: Lamp-Lamp1-Green
    Lamp1 (683,230 29x33), variable: MAIN.M2_SNR2, style: Lamp-Lamp1-Green
    Lamp1 (432,227 29x33), variable: MAIN.M1_sNR, style: Lamp-Lamp1-Green
    Lamp1 (946,225 29x33), variable: MAIN.M3_SNR2, style: Lamp-Lamp1-Green
    Lamp1 (775,225 29x33), variable: MAIN.M3_SNR1, style: Lamp-Lamp1-Green
    Lamp1 (861,298 29x33), variable: MAIN.M3_SNR3, style: Lamp-Lamp1-Green
    Rectangle (769,651 70x27), "%s", text variable: MAIN.show_CG1
    Rectangle (466,70 71x29), "%s", text variable: MAIN.show_CG2
    Rectangle (726,69 71x29), "%s", text variable: MAIN.show_CG3
    ImageSwitcher (653,226 21x32), variable: MOTION.LM_GoRight, input disabled if: MOTION.LM_GoLeft, background image: ImagePool_Base.RIGHT_ON, image: ImagePool_Base.RIGHT_OFF, behaviour: TOGGLE
    ImageSwitcher (812,227 20x29), variable: MOTION.RM_GoLeft, input disabled if: MOTION.RM_GoRight, background image: ImagePool_Base.LEFT_ON, image: ImagePool_Base.LEFT_OFF, behaviour: TOGGLE
    ImageSwitcher (925,230 21x32), variable: MOTION.RM_GoRight, input disabled if: MOTION.RM_GoLeft, background image: ImagePool_Base.RIGHT_ON, image: ImagePool_Base.RIGHT_OFF, behaviour: TOGGLE
    ImageSwitcher (554,227 22x34), variable: MOTION.LM_GoLeft, input disabled if: MOTION.LM_GoRight, background image: ImagePool_Base.LEFT_ON, image: ImagePool_Base.LEFT_OFF, behaviour: TOGGLE
    Textfield (577,71 71x29), "%3.1f", text variable: MAIN.ATM1_dis
    Textfield (846,69 71x29), "%3.1f", text variable: MAIN.ATM2_dis
    Textfield (954,639 64x30), "%3.1f", text variable: MAIN.ATM3_dis
    Textfield (29,503 70x30), "%3.1f", text variable: MAIN.MFC1_dis
    Textfield (30,597 70x30), "%3.1f", text variable: MAIN.MFC2_dis
    Textfield (29,537 70x30), "%3.1f", text variable: MFC1_Inp
        OnMouseClick: write the text variable via Default, min 0, max 1000
    Textfield (30,632 70x31), "%3.1f", text variable: MFC2_Inp
        OnMouseClick: write the text variable via Default, min 0, max 100
    Button (45,156 58x25), "open", input disabled if: GV1_OPN_DEVINP
        tap GV1_btn_open
    Button (110,154 59x27), "close", input disabled if: GV1_CLS_DEVINP
        tap GV1_btn_close
    Button (46,195 58x28), "open"
        tap GV2_btn_open
    Button (109,195 61x28), "close"
        tap GV2_btn_close
    ImageSwitcher (471,208 21x145), variable: DI2_1, background image: ImagePool_Base.GV_OPEN, image: ImagePool_Base.GV_CLS, behaviour: TOGGLE
    ImageSwitcher (735,210 21x145), variable: DI2_3, background image: ImagePool_Base.GV_OPEN, image: ImagePool_Base.GV_CLS, behaviour: TOGGLE
    Rectangle (100,288 67x27), "%s", text variable: MAIN.PV1
    Rectangle (100,323 67x27), "%s", text variable: MAIN.PV2
    Rectangle (100,361 67x27), "%s", text variable: MAIN.PV3
    Button (954,718 64x30), "LV80"
        toggle GVL.lv80_btn
    Button (954,679 64x30), "WSU251", input disabled if: MAIN.WSU_DEVINP
        toggle GVL.WSU_btn
    Lamp1 (847,722 27x32), variable: DI1_4, style: Lamp-Lamp1-Green
    Textfield (555,562 70x30), "%d", text variable: GVL.HTC_SetPr
        OnMouseClick: write the text variable via Default, min 0, max 300
    Textfield (639,561 70x30), "%d", text variable: GVL.HTC_SetPos
        OnMouseClick: write the text variable via Default, min 0, max 1000
    Rectangle (555,603 70x30), "%d", text variable: MAIN.HTC_ReadPr
    Rectangle (639,603 70x30), "%d", text variable: MAIN.HTC_ReadPos
    Button (555,644 70x30)
        toggle DO4_6
    Button (30,481 70x20)
        toggle mfc1_open_btn
    Button (30,573 70x20)
        toggle mfc2_open_btn
    Button (557,503 71x30), "%s", text variable: MAIN.cur_mode
        toggle MAIN.HTC_MODE_Pr
    Button (225,399 43x25), "UP"
        tap MAIN.m3_pin_up
    Button (276,399 52x25), "DOWN"
        tap MAIN.m3_pin_down
    Button (224,359 43x28), "OPEN"
        tap MAIN.m3_rail_open
    Button (276,359 52x28), "CLOSE"
        tap MAIN.M3_rail_CLOSE
    Lamp1 (188,355 31x37), variable: MAIN.M3_rail_opened, style: Lamp-Lamp1-Yellow
    Lamp1 (330,355 31x37), variable: MAIN.M3_rail_closed, style: Lamp-Lamp1-Yellow
    Lamp1 (188,396 31x37), variable: DI3_4, style: Lamp-Lamp1-Yellow
    Lamp1 (333,396 31x37), variable: DI3_5, style: Lamp-Lamp1-Yellow
    Textfield (30,289 67x25), "%d", text variable: GVL.SV1
        OnMouseClick: write the text variable via Default, min 0, max 300
    Textfield (30,321 67x25), "%d", text variable: GVL.SV2
        OnMouseClick: write the text variable via Default, min 0, max 300
    Button (194,275 111x30), "TAKE UP"
        tap MAIN.m3_up_btn
    Button (194,316 111x30), "PUT DOWN"
        tap MAIN.m3_down_btn
    ImageSwitcher (583,146 37x38), variable: MAIN.ATM1_STS, input disabled if: 1, background image: ImagePool_Base.ATM_ON, image: ImagePool_Base.ATM_OFF, behaviour: TOGGLE
    ImageSwitcher (842,146 37x38), variable: MAIN.ATM2_STS, input disabled if: 1, background image: ImagePool_Base.ATM_ON, image: ImagePool_Base.ATM_OFF, behaviour: TOGGLE
    ImageSwitcher (914,594 37x38), variable: MAIN.ATM3_STS, input disabled if: 1, background image: ImagePool_Base.ATM_ON, image: ImagePool_Base.ATM_OFF, behaviour: TOGGLE
    ImageSwitcher (877,701 73x63), variable: MAIN.LV80_STS, input disabled if: 1, background image: ImagePool_Base.LV80_ON, image: ImagePool_Base.LV80_OFF, behaviour: TOGGLE
    ImageSwitcher (877,660 29x55), variable: MAIN.WSU_STS, input disabled if: 1, background image: ImagePool_Base.WSU_ON, image: ImagePool_Base.WSU_OFF, behaviour: TOGGLE
    ImageSwitcher (880,526 36x36), variable: MAIN.TV_STS, input disabled if: 1, background image: ImagePool_Base.TV_ON, image: ImagePool_Base.TV_OFF, behaviour: TOGGLE
    Button (589,228 42x30)
        tap MOTION.LM_Stop
    Button (853,230 42x30)
        tap MOTION.RM_Stop
    Textfield (681,716 150x31), "%s", text variable: MAIN.cur_time
    Button (312,277 51x67), "RESET"
        tap MAIN.reset_btn
    Lamp1 (117,398 27x32), variable: DI1_6, style: Lamp-Lamp1-Green
    Lamp1 (44,398 27x32), variable: DI1_5, style: Lamp-Lamp1-Green
    Button (194,154 70x30), "Rec Start", colour toggle: GVL.Rec_start_btn
        toggle GVL.Rec_start_btn
    ImageSwitcher (270,537 43x52), variable: DO2_3, background image: ImagePool_Base.VAL_ON, image: ImagePool_Base.VAL_OFF, behaviour: TOGGLE
    ImageSwitcher (270,637 43x52), variable: DO2_4, background image: ImagePool_Base.VAL_ON, image: ImagePool_Base.VAL_OFF, behaviour: TOGGLE
    ImageSwitcher (362,631 43x52), variable: DO2_6, background image: ImagePool_Base.VAL_ON, image: ImagePool_Base.VAL_OFF, behaviour: TOGGLE
    ImageSwitcher (448,633 43x52), variable: DO3_3, background image: ImagePool_Base.VAL_ON, image: ImagePool_Base.VAL_OFF, behaviour: TOGGLE
    Label (532,69 44x30), "torr"
    Label (792,70 44x30), "torr"
    Label (233,549 40x30), "NC4"
    Label (228,647 40x30), "NC5"
    Label (324,643 40x30), "NC7"
    Label (409,643 40x30), "NC12"
    Label (835,651 44x30), "torr"
    Label (643,70 44x30), "KPA"
    Label (915,69 44x30), "KPA"
    Label (590,532 44x30), "(porr)"
    Label (678,534 44x30), "(%)"
    Button (16,716 103x30), "MAIN"
        OnMouseClick: change screen: MainBase
    Button (127,716 103x30), "PARAMETER"
        OnMouseClick: change screen: PARAMETER
    Button (238,716 103x30), "ALARM"
        OnMouseClick: change screen: ALARM
    Button (349,716 103x30), "IO"
        OnMouseClick: change screen: IO_TABLE
    Button (460,716 103x30), "MOTION"
        OnMouseClick: change screen: MOTION
    Button (571,716 103x30), "Recipe"
        OnMouseClick: change screen: Recipt
    Button (277,154 70x30), "Rec Cancel"
        tap Rec_stop_btn
    Textfield (196,193 147x30), "%s", text variable: GVL.CUR_step_name
END_VISUALIZATION

// ---- VISUs/MOTION.TcVIS
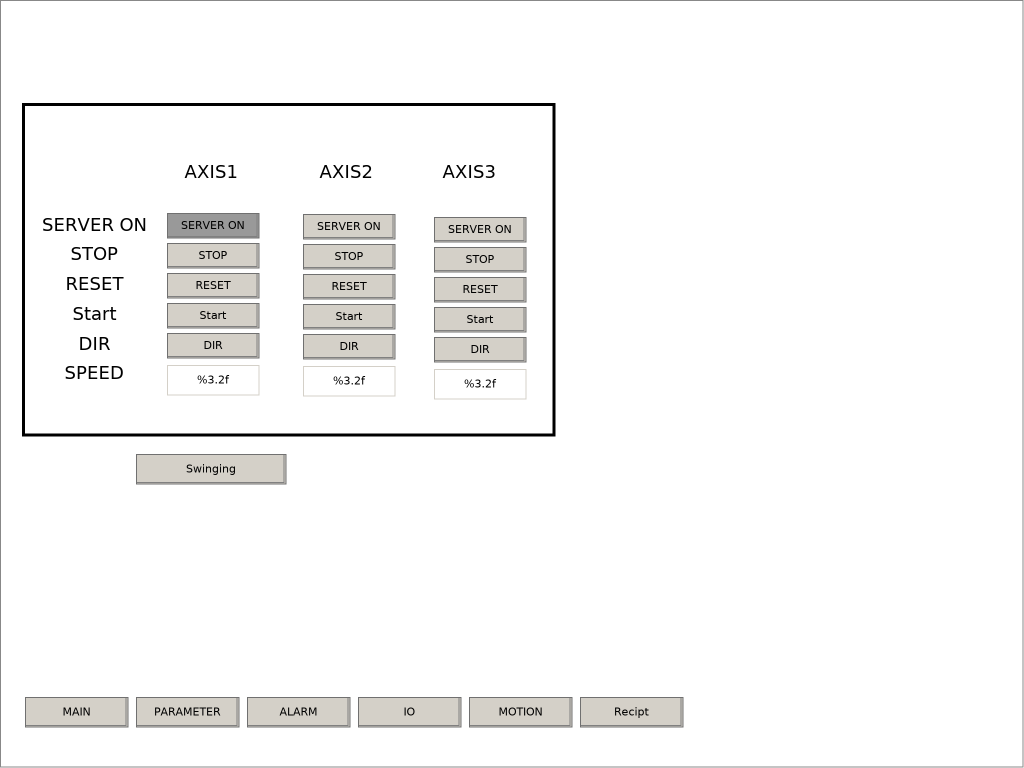
VISUALIZATION MOTION  // 1024x768, background image ImagePool_Base.base
    RoundedRectangle (22,103 533x333)
    Label (14,210 161x30), "SERVER ON"
    Label (14,239 161x30), "STOP"
    Label (14,269 161x30), "RESET"
    Label (14,299 161x30), "Start"
    Label (14,358 161x30), "SPEED"
    Button (167,213 92x25), "SERVER ON"
        toggle MOTION.Pwr_En_1 p2164770859=TRUE
    Button (167,243 92x25), "STOP"
        tap MOTION.stop_1
    Button (167,273 92x25), "RESET"
        tap MOTION.reset_1
    Button (167,303 92x25), "Start"
        tap MOTION.V_ex1
    Textfield (167,365 92x30), "%3.2f", text variable: MOTION.VV1
        OnMouseClick: write the text variable via Default, min 0, max 300
    Button (167,333 92x25), "DIR"
        toggle MOTION.DIR1
    Label (14,329 161x30), "DIR"
    Button (303,214 92x25), "SERVER ON"
        toggle MOTION.Pwr_En_2
    Button (303,244 92x25), "STOP"
        tap MOTION.stop_2
    Button (303,274 92x25), "RESET"
        tap MOTION.reset_2
    Button (303,304 92x25), "Start"
        tap MOTION.V_ex2
    Textfield (303,366 92x30), "%3.2f", text variable: MOTION.VV2
        OnMouseClick: write the text variable via Default, min 0, max 300
    Button (303,334 92x25), "DIR"
        toggle MOTION.DIR2
    Button (434,217 92x25), "SERVER ON"
        toggle MOTION.Pwr_En_3
    Button (434,247 92x25), "STOP"
        tap MOTION.stop_3
    Button (434,277 92x25), "RESET"
        tap MOTION.reset_3
    Button (434,307 92x25), "Start"
        tap MOTION.V_ex3
    Textfield (434,369 92x30), "%3.2f", text variable: MOTION.VV3
        OnMouseClick: write the text variable via Default, min 0, max 300
    Button (434,337 92x25), "DIR"
        toggle MOTION.DIR3 p2164770859=TRUE
    Label (155,157 113x30), "AXIS1"
    Label (290,157 113x30), "AXIS2"
    Label (413,157 113x30), "AXIS3"
    Button (136,454 150x30), "Swinging"
        toggle MOTION.swinging
    Button (25,697 103x30), "MAIN"
        OnMouseClick: change screen: MainBase
    Button (136,697 103x30), "PARAMETER"
        OnMouseClick: change screen: PARAMETER
    Button (247,697 103x30), "ALARM"
        OnMouseClick: change screen: ALARM
    Button (358,697 103x30), "IO"
        OnMouseClick: change screen: IO_TABLE
    Button (469,697 103x30), "MOTION"
        OnMouseClick: change screen: MOTION
    Button (580,697 103x30), "Recipt"
        OnMouseClick: change screen: Recipt
END_VISUALIZATION

// ---- VISUs/PARAMETER.TcVIS
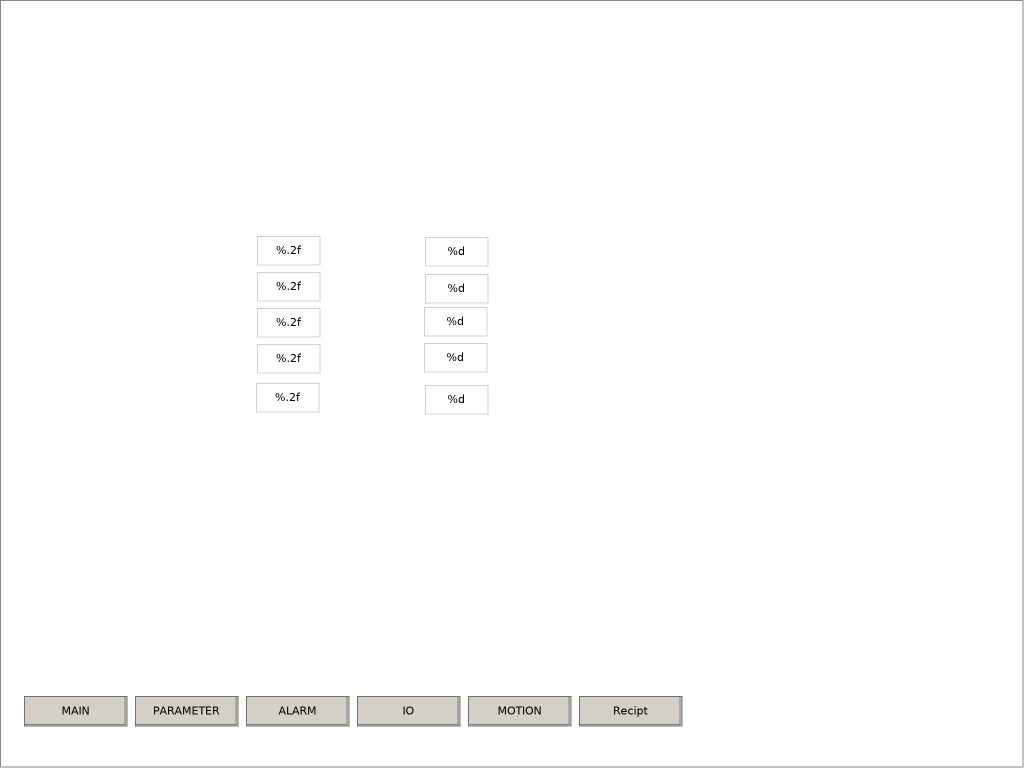
VISUALIZATION PARAMETER  // 1024x768, background image ImagePool_Base.PARAMETER
    Textfield (425,237 63x29), "%d", text variable: MAIN.MFC_delay_show
        OnMouseClick: write the text variable via Default
    Textfield (425,274 63x29), "%d", text variable: MAIN.water_temp_delay_show
        OnMouseClick: write the text variable via Default
    Textfield (424,343 63x29), "%d", text variable: MAIN.WP_delta_delay_show
        OnMouseClick: write the text variable via Default
    Textfield (425,385 63x29), "%d", text variable: MAIN.Heater_temp_delay_show
        OnMouseClick: write the text variable via Default
    Textfield (257,236 63x29), "%.2f", text variable: MAIN.MFC_alarm_setting
        OnMouseClick: write the text variable via Default
    Textfield (257,272 63x29), "%.2f", text variable: MAIN.water_temp_setting
        OnMouseClick: write the text variable via Default
    Textfield (257,308 63x29), "%.2f", text variable: MAIN.WP_delta_setting
        OnMouseClick: write the text variable via Default
    Textfield (257,344 63x29), "%.2f", text variable: MAIN.WP_delta_setting
        OnMouseClick: write the text variable via Default
    Textfield (256,383 63x29), "%.2f", text variable: MAIN.Heater_temp_seeting
        OnMouseClick: write the text variable via Default
    Textfield (424,307 63x29), "%d", text variable: MAIN.WP_delta_delay_show
        OnMouseClick: write the text variable via Default
    Button (24,696 103x30), "MAIN"
        OnMouseClick: change screen: MainBase
    Button (135,696 103x30), "PARAMETER"
        OnMouseClick: change screen: PARAMETER
    Button (246,696 103x30), "ALARM"
        OnMouseClick: change screen: ALARM
    Button (357,696 103x30), "IO"
        OnMouseClick: change screen: IO_TABLE
    Button (468,696 103x30), "MOTION"
        OnMouseClick: change screen: MOTION
    Button (579,696 103x30), "Recipt"
        OnMouseClick: change screen: Recipt
END_VISUALIZATION

// ---- VISUs/Recipt.TcVIS
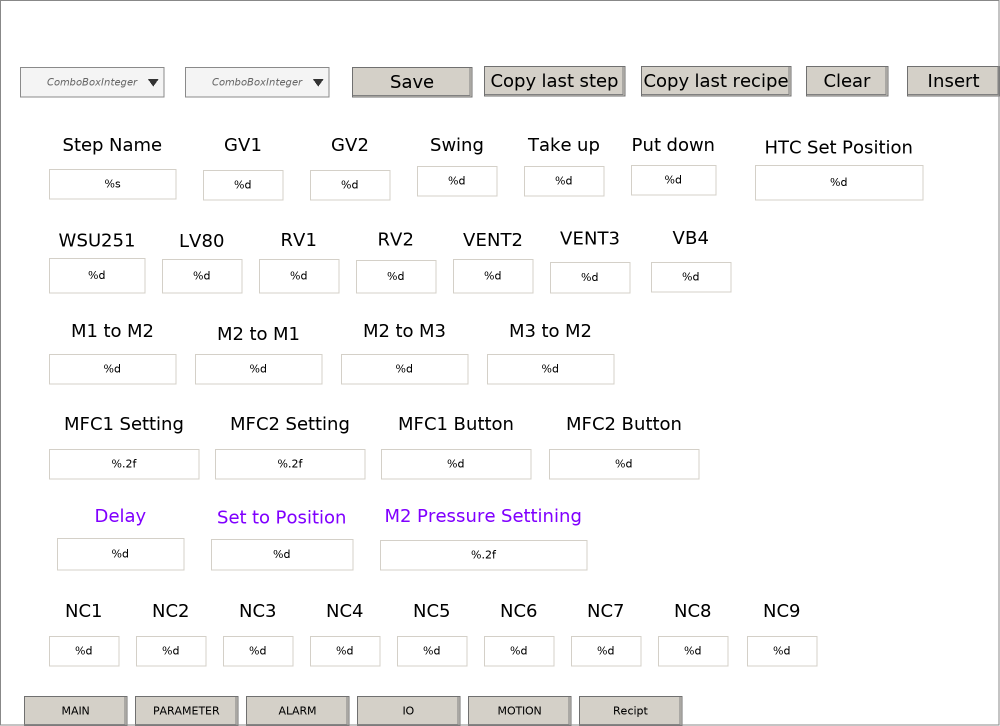
VISUALIZATION Recipt  // 1000x726, background image ImagePool_Base.base
    Button (24,696 103x30), "MAIN"
        OnMouseClick: change screen: MainBase
    Button (135,696 103x30), "PARAMETER"
        OnMouseClick: change screen: PARAMETER
    Button (246,696 103x30), "ALARM"
        OnMouseClick: change screen: ALARM
    Button (357,696 103x30), "IO"
        OnMouseClick: change screen: IO_TABLE
    Button (468,696 103x30), "MOTION"
        OnMouseClick: change screen: MOTION
    Button (579,696 103x30), "Recipt"
        OnMouseClick: change screen: Recipt
    Group (49,409 650x70)
        Group (0,0 150x70)
            Label (0,0 150x30), "MFC1 Setting"
            Textfield (0,40 150x30), "%.2f", text variable: Temp_Recipt_step.MFC1_Setting
                OnMouseClick: write the text variable via Default
        Group (166,0 150x70)
            Label (0,0 150x30), "MFC2 Setting"
            Textfield (0,40 150x30), "%.2f", text variable: Temp_Recipt_step.MFC2_Setting
                OnMouseClick: write the text variable via Default
        Group (332,0 150x70)
            Label (0,0 150x30), "MFC1 Button"
            Textfield (0,40 150x30), "%d", text variable: Temp_Recipt_step.MFC1_button
                OnMouseClick: write the text variable via Default, min 0, max 1
        Group (500,0 150x70)
            Label (0,0 150x30), "MFC2 Button"
            Textfield (0,40 150x30), "%d", text variable: Temp_Recipt_step.MFC2_button
                OnMouseClick: write the text variable via Default, min 0, max 1
    ComboBoxInteger (185,67 144x30), variable: MAIN.cur_step, text list: 'step'
    ComboBoxInteger (20,67 144x30), variable: MAIN.cur_Rec, text list: 'Recipt_no'
    Button (352,67 120x30), "Save"
        tap MAIN.save_step_btn
    Group (49,596 768x70)
        Label (0,0 70x30), "NC1"
        Textfield (0,40 70x30), "%d", text variable: Temp_Recipt_step.NC1
            OnMouseClick: write the text variable via Default, min 0, max 1
        Label (87,0 70x30), "NC2"
        Textfield (87,40 70x30), "%d", text variable: Temp_Recipt_step.NC2
            OnMouseClick: write the text variable via Default, min 0, max 1
        Label (174,0 70x30), "NC3"
        Textfield (174,40 70x30), "%d", text variable: Temp_Recipt_step.NC3
            OnMouseClick: write the text variable via Default, min 0, max 1
        Label (261,0 70x30), "NC4"
        Textfield (261,40 70x30), "%d", text variable: Temp_Recipt_step.NC4
            OnMouseClick: write the text variable via Default, min 0, max 1
        Label (348,0 70x30), "NC5"
        Textfield (348,40 70x30), "%d", text variable: Temp_Recipt_step.NC5
            OnMouseClick: write the text variable via Default, min 0, max 1
        Label (435,0 70x30), "NC6"
        Textfield (435,40 70x30), "%d", text variable: Temp_Recipt_step.NC6
            OnMouseClick: write the text variable via Default, min 0, max 1
        Label (522,0 70x30), "NC7"
        Textfield (522,40 70x30), "%d", text variable: Temp_Recipt_step.NC7
            OnMouseClick: write the text variable via Default, min 0, max 1
        Label (609,0 70x30), "NC8"
        Textfield (609,40 70x30), "%d", text variable: Temp_Recipt_step.NC8
            OnMouseClick: write the text variable via Default, min 0, max 1
        Label (698,0 70x30), "NC9"
        Textfield (698,40 70x30), "%d", text variable: Temp_Recipt_step.NC9
            OnMouseClick: write the text variable via Default, min 0, max 1
    Group (49,316 565x70)
        Group (0,0 127x70)
            Label (0,0 127x30), "M1 to M2"
            Textfield (0,38 127x30), "%d", text variable: Temp_Recipt_step.M1toM2
                OnMouseClick: write the text variable via Default, min 0, max 1
        Group (146,3 127x67)
            Label (0,0 127x30), "M2 to M1"
            Textfield (0,35 127x30), "%d", text variable: Temp_Recipt_step.M2toM1
                OnMouseClick: write the text variable via Default, min 0, max 1
        Group (292,0 127x70)
            Label (0,0 127x30), "M2 to M3"
            Textfield (0,38 127x30), "%d", text variable: Temp_Recipt_step.M2toM3
                OnMouseClick: write the text variable via Default, min 0, max 1
        Group (438,0 127x70)
            Label (0,0 127x30), "M3 to M2"
            Textfield (0,38 127x30), "%d", text variable: Temp_Recipt_step.M3toM2
                OnMouseClick: write the text variable via Default, min 0, max 1
    Button (484,66 141x30), "Copy last step"
        tap MAIN.Copy_step
    Button (641,66 150x30), "Copy last recipe"
        tap MAIN.Copy_recipe
    Button (806,66 82x30), "Clear"
        tap MAIN.clear_step_btn
    Group (49,130 874x70)
        Group (0,0 127x70)
            Label (0,0 127x30), "Step Name"
            Textfield (0,39 127x30), "%s", text variable: Temp_Recipt_step.step_Name
                OnMouseClick: write the text variable via Default
        Group (154,0 80x70)
            Label (0,0 80x30), "GV1"
            Textfield (0,40 80x30), "%d", text variable: Temp_Recipt_step.GV1
                OnMouseClick: write the text variable via Default, min 0, max 1
        Group (261,0 80x70)
            Label (0,0 80x30), "GV2"
            Textfield (0,40 80x30), "%d", text variable: Temp_Recipt_step.GV2
                OnMouseClick: write the text variable via Default, min 0, max 1
        Textfield (706,35 168x35), "%d", text variable: Temp_Recipt_step.Position_setting
            OnMouseClick: write the text variable via Default
        Label (706,0 168x35), "HTC Set Position"
        Group (368,0 80x70)
            Label (0,0 80x30), "Swing"
            Textfield (0,36 80x30), "%d", text variable: Temp_Recipt_step.Swing
                OnMouseClick: write the text variable via Default, min 0, max 1
        Group (475,0 80x70)
            Textfield (0,36 80x30), "%d", text variable: Temp_Recipt_step.Take_up
                OnMouseClick: write the text variable via Default, min 0, max 1
            Label (0,0 80x30), "Take up"
        Group (582,0 92x70)
            Textfield (0,35 85x30), "%d", text variable: Temp_Recipt_step.Put_down
                OnMouseClick: write the text variable via Default, min 0, max 1
            Label (0,0 85x30), "Put down"
    Group (57,500 530x70)
        Group (154,2 142x68)
            Textfield (0,37 142x31), "%d", text variable: Temp_Recipt_step.Set2Pos
                OnMouseClick: write the text variable via Default, min 0, max 1
            Label (0,0 142x31), "Set to Position"
        Group (323,1 207x69)
            Label (0,0 207x30), "M2 Pressure Settining"
            Textfield (0,39 207x30), "%.2f", text variable: Temp_Recipt_step.M2_pressure_setting
                OnMouseClick: write the text variable via Default
        Group (0,0 127x70)
            Label (0,0 127x32), "Delay"
            Textfield (0,38 127x32), "%d", text variable: Temp_Recipt_step.delay
                OnMouseClick: write the text variable via Default
    Group (49,223 682x70)
        Group (602,0 80x69)
            Textfield (0,39 80x30), "%d", text variable: Temp_Recipt_step.VB4
                OnMouseClick: write the text variable via Default, min 0, max 1
            Label (0,0 80x30), "VB4"
        Group (404,0 80x70)
            Label (0,0 80x34), "VENT2"
            Textfield (0,36 80x34), "%d", text variable: Temp_Recipt_step.VENT2
                OnMouseClick: write the text variable via Default, min 0, max 1
        Group (210,0 80x70)
            Label (0,0 80x34), "RV1"
            Textfield (0,36 80x34), "%d", text variable: Temp_Recipt_step.RV1
                OnMouseClick: write the text variable via Default, min 0, max 1
        Group (307,0 80x70)
            Label (0,0 80x33), "RV2"
            Textfield (0,37 80x33), "%d", text variable: Temp_Recipt_step.RV2
                OnMouseClick: write the text variable via Default, min 0, max 1
        Group (0,0 96x70)
            Label (0,0 96x35), "WSU251"
            Textfield (0,35 96x35), "%d", text variable: Temp_Recipt_step.WSU251
                OnMouseClick: write the text variable via Default, min 0, max 1
        Group (113,0 80x70)
            Label (0,0 80x36), "LV80"
            Textfield (0,36 80x34), "%d", text variable: Temp_Recipt_step.LV80
                OnMouseClick: write the text variable via Default, min 0, max 1
        Group (501,0 80x70)
            Textfield (0,39 80x31), "%d", text variable: Temp_Recipt_step.VENT3
                OnMouseClick: write the text variable via Default, min 0, max 1
            Label (0,0 80x31), "VENT3"
    Button (907,66 93x30), "Insert", colour toggle: MAIN.insert_btn
        toggle MAIN.insert_btn
END_VISUALIZATION
